// TwinCAT 3 PLC project PLC_Portale
// Title: TFPalletizer
// Author: Pugnaghi
// libraries:
//   Tc2_Math, * (Beckhoff Automation GmbH)
//   Tc2_MC2, * (Beckhoff Automation GmbH)
//   Tc2_MC2_Drive, * (Beckhoff Automation GmbH)
//   Tc2_Standard, * (Beckhoff Automation GmbH)
//   Tc2_SUPS, * (Beckhoff Automation GmbH)
//   Tc2_System, * (Beckhoff Automation GmbH)
//   Tc2_Utilities, * (Beckhoff Automation GmbH)
//   Tc3_Module, * (Beckhoff Automation GmbH)
//   Tc3_Standard, * (Beckhoff Automation GmbH)
//   TFDataLogger, * (Tecnoferrari)
//   TFInterpolazioneAssi, * (TecnoFerrari)
//   TFPLC, * (Tecnoferrari)
//   TF_CambioProduzioneLinea, * (Tecnoferrari)
//   TF_Ovem, * (Tecnoferrari)
// project tree:
//   Data types/AlbertoPruevas/BloqueFunciones/CalculoFormaciones/ Fb_CalculoCoordenadasFinalesFormacion.TcPOU, Fb_CalculoTodo180CoordenadasFinales.TcPOU, Fb_Fb_CalculoTodo0CoordenadasFinales.TcPOU
//   Data types/AlbertoPruevas/BloqueFunciones/ Fb_SensoresTasteggio.TcPOU
//   Data types/AlbertoPruevas/Enumeraciones/ E_Ul_RecogidaCaballete.TcDUT
//   Data types/AlbertoPruevas/Estructuras/Es_FormacionCaballete/EstructuraCaballetePiking/ ES_DatosPosCaballete.TcDUT, Es_PiezasCaballetePiking.TcDUT
//   Data types/AlbertoPruevas/Estructuras/Es_FormacionCaballete/ Es_CoordenadasCaballeteLadoA.TcDUT, Es_CoordenadasCaballeteLadoA_ladoB.TcDUT, Es_CoordenadasCaballeteLadoB.TcDUT, ES_dimensionPiezaLadoA_ladoB.TcDUT, Es_NumeroPiezasCaballete.TcDUT, ES_SpesoreLastra_A_B.TcDUT
//   Data types/AlbertoPruevas/Estructuras/ Es_Ingombro_PorPosicion.TcDUT (not stored), Es_LadosCaballete.TcDUT, Es_PiezasCaballete.TcDUT, ProgramaEjecucion.TcDUT
//   Data types/AlbertoPruevas/Funciones/FuncionesFormaciones/ Fun_CalculoCoordenadasFinalesFormacion.TcPOU
//   Data types/AlbertoPruevas/Funciones/ FunLadoTrabajoCaballete.TcPOU, Fun_NumeroPiezasLadoCaballete.TcPOU, Fun_PiezaLadoCaballete.TcPOU, Fun_SensoresTasteggio.TcPOU
//   Data types/DatiVari/EAP/ ST_EAPAxeState.TcDUT, ST_EAPCylinderState.TcDUT, ST_EAPMachineState.TcDUT, ST_EAPModuleState.TcDUT, ST_EAPOvemStatus.TcDUT, ST_EAPPinzaVenstoseStateComplete.TcDUT, ST_EAPPinzaVentoseDeviceState.TcDUT, ST_EAPStatoPortaleVisu.TcDUT
//   Data types/DatiVari/ e_StatoMacchinaWMS.TcDUT, e_SupportTypeAriostea.TcDUT, ST_HskFromSupervisor.TcDUT, ST_HskToSupervisor.TcDUT, ST_StatisticData.TcDUT, ST_SupervisorData.TcDUT
//   Data types/DatiVari/Workorder/ ST_DataWorkArea.TcDUT, ST_DimensionElement.TcDUT, ST_LayerData.TcDUT, ST_SlabData.TcDUT, ST_SupportData.TcDUT, ST_WorkOrder.TcDUT, ST_WorkOrder_Premium.TcDUT
//   Data types/Enum/ e_Disposizione_FTC_WA.TcTLEO, e_Disposizione_Postazioni.TcDUT, e_PosizionePinza.TcDUT, e_RiferimentoPostazione.TcTLEO, e_OrdinamentoPostazione.TcTLEO, e_StatoWorkOrder.TcDUT, e_Stato_Apprendimento.TcTLEO, e_Stato_ElementoLista.TcTLEO, e_Stato_Missione.TcTLEO, e_Stato_PickPoint.TcTLEO, e_Stato_Pareggiatura_Lastra.TcTLEO, e_Stato_LetturaBarCode.TcTLEO, e_Stato_Prodotto_Su_PickPoint.TcTLEO, e_Stato_Prelievo.TcTLEO, e_Stato_Ingombro_EE.TcTLEO, e_Stato_Layer.TcTLEO, e_Stato_Prodotto_Generico.TcTLEO, e_Stato_WAManager.TcTLEO, e_Priorita_PickPoint.TcTLEO, e_Stato_WorkArea.TcTLEO, e_Stato_ListaDiProduzione.TcTLEO, e_TipologiaAreaLaser.TcDUT, e_Tipologia_Rul_Prel.TcDUT, e_Tipo_Elemento_Da_Lavorare.TcDUT, e_Tipo_Magazzino_Falde.TcTLEO, e_Tipo_ChiusuraAsseK.TcTLEO, e_Tipo_Funzionamento.TcTLEO, e_Tipo_WorkArea.TcTLEO, e_Tipo_Ribaltino.TcTLEO, e_Tipo_PickPoint.TcTLEO, e_Tipo_Falda.TcTLEO, e_Tipo_Pallet.TcTLEO, e_Tipo_PresaEndEffector.TcTLEO, e_Tipo_Traiettoria.TcTLEO, e_Verso_Pallettizzatore.TcTLEO
//   Data types/Enum/Formatura/ e_TipologiaDeposito.TcDUT
//   Data types/Enum/Trasporti/ e_ElementZone.TcDUT, e_PosizioneRullieraMobile.TcDUT, e_StatoCentratura.TcDUT, e_TipoMacchinaTrasporti.TcDUT
//   Data types/LGV/ e_Tipo_Richiesta_LGV.TcTLEO, e_Stato_Richiesta_LGV_1.TcTLEO, LGV_Stato_Formatura.TcDUT, LGV_Stato_Pallettizzatore.TcDUT, LGV_Stato_Postazione.TcDUT, e_Stato_Operazione_LGV.TcTLEO
//   Data types/Nuove/ ST_OffsetAllDirection.TcDUT, TFMachinePalletizer_ListaProduzione_WAM_HMI.TcDUT, TFMachinePalletizer_WorkAreaTransport_State.TcDUT, TFMachinePalletizer_WorkPlacePointToPalletizer.TcDUT, TFMachinePalletizer_WorkPlacePointFromPalletizer.TcDUT, TFCodiciPerFormatura.TcDUT, TFError_WAM.TcDUT, TFMachinePalletizer_DataElementMP.TcDUT, TFMachinePalletizer_PinzaVentoseManCmd.TcDUT, TFMachinePalletizer_ApprendimentoQuota.TcDUT, TFMachinePalletizer_CoordinateApprendimento.TcDUT, TFMachinePalletizer_LatoApprendimento.TcDUT, TFMachinePalletizer_DataElement.TcDUT, TFMachinePalletizer_EndEffector.TcDUT, TFMachinePalletizer_BarCode.TcDUT, TFMachinePalletizer_ListaProduzione.TcDUT, TFMachinePalletizer_ListaProduzione_WAM.TcDUT, TFMachinePalletizer_OffsetElement.TcDUT, TFMachinePalletizer_PickPlaceParameters.TcDUT, TFMachinePalletizer_PinzaState.TcDUT, TFMAchinePalletizer_PinzaVentoseStatus.TcDUT, TFMachinePalletizer_PinzaVentose_OUT.TcDUT, TFMachinePalletizer_PlaceElement.TcDUT, TFMachinePalletizer_PlaceElementList.TcDUT, TFMachinePalletizer_WorkPickPointOffset.TcDUT, TFMachinePalletizer_WorkPickPoint_State.TcDUT, TFMachinePalletizer_WorkPickPointRoller_State_DaLinea.TcDUT, TFMachinePalletizer_WorkPickPointRoller_State_ALinea.TcDUT, TFMachinePalletizer_WorkPickPointStore_State.TcDUT, TFMachinePalletizer_WorkPickPointSlab.TcDUT, TF_CylinderState.TcDUT, TFMchinePalletizer_PinzaVentose_IN.TcDUT, TFPalletizerModules.TcDUT
//   Data types/Picking/ e_TypologySupDataPicking.TcDUT, ST_DataManualPicking.TcDUT, ST_WorkAreaDataPicking.TcDUT
//   Data types/Programmi Movimento/ TFModulePortaleStatus.TcDUT, AxHomingParameters.TcDUT, Ax_Palletizer_Basic_Parameters.TcDUT, Ax_Palletizer_Nominal_Parameters.TcDUT, GestioneEncoderEsterno.TcDUT, MissionStateCase.TcDUT, Module_Palletizer_Aspirazione_IN.TcDUT, Module_Palletizer_Aspirazione_ManCmd.TcDUT, Module_Palletizer_AX_OUT.TcDUT, Module_Palletizer_AX_IN.TcDUT, Ax_Program_Parameters.TcDUT, Descrittore_Programma.TcDUT, Ax_Palletizer_Parameters.TcDUT, Module_Palletizer_Aspirazione_OUT.TcDUT, OffsetSicurezzaIngombro.TcDUT, OffsetDistacco.TcDUT, Offset_Pass_Mode.TcDUT, Offset_Prelievi_Lenti.TcDUT, Offeset_Apprendimento.TcDUT, Offset_Sicurezza.TcDUT, Offset_Sicurezza_Anticipo_Movimenti.TcDUT, Overide_Dinamico.TcDUT, ProgrammaLog.TcDUT, Stato_Ciclo_Lavoro.TcDUT, StrutturaGenericaQuotaAssi.TcDUT, TFDimensioniPinza.TcDUT, TFMachinePalletizer_ModuleState.TcDUT, TFMachinePalletizer_MachineState.TcDUT, TFMachinePalletizer_VelocityOverride_TF.TcDUT, TFModulePalletizerRobot_Point_TF.TcDUT, TFModulePalletizerSTATUS_TF.TcDUT, TFTraiettoria.TcDUT, TFWorkAreaManager.TcDUT, Work_PickPoint_Dimension.TcDUT
//   Data types/ StatoPostazioneHMI.TcDUT, StatoLineaDepal.TcDUT, TFDatiDaLineaAPal.TcDUT, TFSlab.TcDUT
//   Data types/Programmi Movimento/Enum Programmi/ e_ProgrammiMovimentoX.TcTLEO, e_ProgrammiMovimentoJ.TcTLEO, e_ProgrammiMovimentoY.TcTLEO, e_ProgrammiMovimentoZ.TcTLEO
//   Data types/Scambio Dati Trasporti/ DUT_ArrayPacchi.TcDUT, DUT_Lista_Pacchi_In_Pila.TcDUT, DUT_Struttura_Dati_Pacco.TcDUT
//   Data types/Strutture Aggiornate/ TFMachinePalletizer_FormingForSlab.TcDUT, TFMachinePalletizer_Layer.TcDUT, TFMachinePalletizer_Mission.TcDUT, TFMachinePalletizer_Pallet.TcDUT, TFMachinePalletizer_PalletSlabOld.TcDUT, TFMachinePalletizer_WorkAreaState_VECCHIO.TcDUT, TFMachinePalletizer_WorkAreaState.TcDUT, TFMachinePalletizer_WorkArea.TcDUT, TFMachinePalletizer_WorkPickPoint.TcDUT, TFMachinePalletizer_WorkArea_VECCHIO.TcDUT, TFMachinePalletizer_FormingPack.TcDUT
//   Data types/TF/Aggiornate_20230504/ ST_BarcodeReaderReply.TcDUT, ST_BarcodeReaderRequest.TcDUT, ST_MachinePalletizerAxeManCmd.TcDUT, ST_MachinePalletizerAxeState.TcDUT, ST_MachinePalletizerMachineState.TcDUT, ST_MachinePalletizerModuleState.TcDUT, ST_MachinePalletizerPinzaDeviceState.TcDUT, ST_MachinePalletizerPinzaStateComplete.TcDUT, ST_MachinePalletizerPinzaVentoseManCmd.TcDUT, ST_StatoPostazioneHMI.TcDUT
//   Data types/TF/Barcode/ BarcodeStatus.TcDUT, InputDataLogic.TcDUT, InputKeyence.TcDUT, OutputDataLogic.TcDUT, OutputKeyence.TcDUT, StatusDataLogic.TcDUT, ST_ManCmdBarcode.TcDUT, TFDeviceBCStatus.TcDUT
//   Data types/TF/Handling/ TFHandlingPack.TcDUT
//   Data types/TF/Palletizer/ TFMachinePalletizer_AxeState_TF.TcDUT, TFMachinePalletizer_AxeState_weintek.TcDUT, TFMachinePalletizer_GatesAccess.TcDUT, TFMachinePalletizer_ManCmd.TcDUT, TFMachinePalletizer_ParametersFromHMI.TcDUT, TFMachinePalletizer_WorkAreaOffset.TcDUT, TFMachinePalletizer_WorkAreaSort.TcDUT, TFMachinePalletizer_WorkAreaZone.TcDUT, TFMachinePalletizer_WorkPickPointState_OLD.TcDUT, TFMachinePalletizer_WorkPPOffset.TcDUT, TFMachinePalletizer_Zone.TcDUT, TFModulePalletizerRobot_TCPPar.TcDUT, TFModulePalletizerRobot_Point.TcDUT, TFModulePalletizerRobot_ManCmd.TcDUT, TFMachinePalletizer_AxeParameters.TcDUT, TFMachinePalletizer_AxeManCmd.TcDUT, TFMachinePalletizer_AxeState.TcDUT, TFModulePalletizerRobot_AxisPar.TcDUT, TFMachinePalletizer_Forming_OLD.TcDUT, TFMachinePalletizer_FormingPack_OLD.TcDUT, TFMachinePalletizer_IN.TcDUT, TFMachinePalletizer_Layer_OLD.TcDUT, TFMachinePalletizer_OUT.TcDUT, TFMachinePalletizer_Pallet_OLD.TcDUT, TFMachinePalletizer_VelocityOverride.TcDUT, TFMachinePalletizer_WorkArea_OLD.TcDUT, TFMachinePalletizer_WorkFootprint.TcDUT, TFMachinePalletizer_WorkPickPoint_OLD.TcDUT, TFMachinePalletizer_WorkSpace.TcDUT, TFModulePalletizerRobot_Status.TcDUT, TFModulePalletizerRobot_IN.TcDUT, TFModulePalletizerRobot_OUT.TcDUT
//   Data types/TF/Rulliere/Macchina/ TFMachineTransportIN.TcDUT, TFMachineTransportManCmd.TcDUT, TFMachineTransportOUT.TcDUT
//   Data types/TF/Rulliere/Moduli/Cinghia/ TFCinghiaManCmd.TcDUT, TFCinghia_IN.TcDUT, TFBancoScelta_IN.TcDUT, TFCinghia_OUT.TcDUT, TFCinghiaParameters.TcDUT, TFBancoScelta_OUT.TcDUT, TFMoveParAXCinghia.TcDUT
//   Data types/TF/Rulliere/Moduli/RullieraPallet/ TFAxCentratoreManCmd.TcDUT, TFAxTraslazioneRulliera.TcDUT, TFCentratoreManCmd.TcDUT, TFCentratoreParameters.TcDUT, TFCentratoreStatus.TcDUT, TFCentratore_IN.TcDUT, TFCentratore_OUT.TcDUT, TFMoveParAXCentratore.TcDUT, TFMoveParAXRulliera.TcDUT, TFMoveParAXTraslazioneRulliera.TcDUT, TFRullieraManCmd.TcDUT, TFRullieraMobileManCmd.TcDUT, TFRullieraMobileStatus.TcDUT, TFRullieraParameters.TcDUT, TFRullieraStatus.TcDUT, TFRulliera_IN.TcDUT, TFRulliera_OUT.TcDUT, TFTraslazioneRullieraParameters.TcDUT, TFTraslazioneRulliera_IN.TcDUT
//   Data types/TF/Rulliere/Moduli/ TFAxManCmd.TcDUT, TFAxParameters.TcDUT, TFPortaStatus.TcDUT, TFPortaManCmd.TcDUT, TFGestioneFTC_Misura_OUT.TcDUT, TFBarcodeStatus.TcDUT, TFTransportModules.TcDUT, TFTransportModuleStatus.TcDUT
//   Data types/TF/Rulliere/ TFDimensionElement.TcDUT, TFMachinePalletizer_Pallet_Weintek.TcDUT, TFMachineTransportElement.TcDUT, TFMachineTransportElementWeintek.TcDUT, TFMachineTransport_GatesAccess.TcDUT
//   Global Variables/BarCode/ BarCODE.TcGVL
//   Global Variables/ Comandi_1.TcGVL, Safety.TcGVL, TFMachinesErrors.TcGVL, TFMachinePalletizerVariables.TcGVL, TFMachinePalletizerErrors.TcGVL, TFCmdStates.TcGVL, TFUpsVariables.TcGVL, TO_HMI.TcGVL
//   Global Variables/Configurazione Impianto/ Configurazione_Impianto.TcGVL
//   Global Variables/Errori/ Errori_BarCODE.TcGVL, Errori_CalcoloFormatura.TcGVL, Errori_WAManager.TcGVL
//   Global Variables/TFVariable/ DATA_LOGGER.TcGVL, Dati_Per_Linea.TcGVL, FROM_HMI_PAL.TcGVL, HMI_COMMAND_PAL.TcGVL, HMI_Formatura.TcGVL, IO_TRASPORTI.TcGVL, IO_Virtuali.TcGVL, LGV_Data.TcGVL, Picking.TcGVL, Pinza.TcGVL, QE_BORDO.TcGVL, QE_TERRA.TcGVL, Supervisor_Variable.TcGVL, TFGlobal.TcGVL, TFMotion_Program.TcGVL, TF_CambioProduzione.TcGVL
//   / GlobalTextList.TcGTLO, Plc_Portale.TcTTO, Visualization Manager.TcVMO (not stored)
//   POUs/Check/ CheckBounds.TcPOU, CheckDivDInt.TcPOU, CheckDivLInt.TcPOU, CheckDivLReal.TcPOU, CheckDivReal.TcPOU, CheckLRangeSigned.TcPOU, CheckLRangeUnsigned.TcPOU, CheckPointer.TcPOU, CheckRangeSigned.TcPOU, CheckRangeUnsigned.TcPOU
//   POUs/TFCicliDiLavoro/Lastre/Cicli Depallettizzatore/ TFCiclo_Deposito_Falda_Depal.TcPOU, TFCiclo_Deposito_Lastra_Depal.TcPOU, TFCiclo_Prelievo_Lastra_Depal.TcPOU
//   POUs/TFCicliDiLavoro/Lastre/Cicli di Deposito Lastre/ TFCiclo_Deposito_Falda.TcPOU, TFCiclo_Deposito_Lastra.TcPOU
//   POUs/TFCicliDiLavoro/Lastre/Cicli di Prelievo Lastre/ TFCiclo_Prelievo_Falda.TcPOU, TFCiclo_Prelievo_Lastra.TcPOU
//   POUs/TFCicliDiLavoro/Lastre/ TFCiclo_Di_Riposo_Lastre.TcPOU
//   POUs/TFCicliDiLavoro/ProgrammiMovimento/ TFProgramma_Ciclo_Falda_Lastre.TcPOU, TFProgramma_Ciclo_Lastra.TcPOU, TFProgramma_Ciclo_Riposo_Lastre.TcPOU
//   POUs/TFGateAccess/ TFGateAccess.TcPOU, TFGateAccessDoppiaMacchina.TcPOU, TFGateAccessNoStop.TcPOU
//   POUs/TFLGV/ GateAccessLGV.TcPOU, TFLGV.TcPOU, TFLGV_NEW.TcPOU
//   POUs/TFMachines/ TFMachinePalletizer_TF.TcPOU
//   POUs/TFMachines/Utility/ TFIsWorkflowError.TcPOU, TFIsWorkflowDisableOrEndedOrError.TcPOU, TFWorkflowsAllEnableOrDisable.TcPOU, TFWorkflowsCheckState.TcPOU
//   POUs/TFModules/DataBase/ Record_From_DB.TcDUT, StoredProcedureState.TcDUT, TFSPRicavaDatiDaBarcodeUDC.TcPOU, TFSPRichiestaIngressoMateriale.TcPOU, TFVerificaLetturaBarcodeConDatiDB.TcPOU
//   POUs/TFModules/Misurazione Ingresso/Keyence/ Keyence_LRTB2000C.TcPOU
//   POUs/TFModules/Misurazione Ingresso/ TFGestioneFTC_Misura.TcPOU, TFGestioneFTC_Misura_IN.TcDUT
//   POUs/TFModules/Moduli TF/ TFModulePalletizer_Aspirazione.TcPOU, TFModulePalletizer_AxJ_Lastre.TcPOU, TFModulePalletizer_Pinza.TcPOU, TFModulePalletizer_Pinza_mag.TcPOU, TFModulePalletizer_Pinza_2Ovem.TcPOU, TFModulePalletizer_Ax.TcPOU, TFModulePalletizer_Pinza_Semplice.TcPOU, TFProgramLogUpdate.TcPOU
//   POUs/TFModules/Utility/ TFClearAllCmdModulePinza.TcPOU, TFClearAllCmdModulePinzaCompleta.TcPOU, TFCylinder_ClearAllCommand.TcPOU, TFOVEMClearAllCommand.TcPOU, TFCylinder_HasCommand.TcPOU (excluded from build), TFPalletizerModulesCheckPowerActive.TcPOU, TFPalletizerModulesCommandSend.TcPOU, TFPalletizerModulesCheckState.TcPOU, TFPalletizerIsModuleError.TcPOU
//   POUs/TFPalletizerDataTF/FunzionePerNuovaGestioneTrasporti/ TFNumeroPacchiSuLinea.TcPOU, TFNumeroUltimi_N_TrasportiOccupati.TcPOU, TFPackCodePresenteInWAJolly.TcPOU (excluded from build), TFPackCodePresenteInZona.TcPOU (excluded from build), TFPackCodePresenteInZona_old.TcPOU (excluded from build)
//   POUs/TFPalletizerDataTF/NON_USATE/ TFCalcoliFuoriIngombriColonne.TcPOU (excluded from build), TFCalcoliFuoriIngombriColonne_old.TcPOU (excluded from build), TFCodicePaccoPresenteInFormatura.TcPOU (excluded from build), TFCodicePaccoPresenteInFormaturaAll.TcPOU (excluded from build), TFDepositoContinuoPalletConsentito.TcPOU (excluded from build), TFNumeroPacchiSuLinea_OLD.TcPOU (excluded from build), TFNumeroUltimi_N_TrasportiOccupati_OLD.TcPOU (excluded from build), TFPalletizerWorkAreaManagerTF.TcPOU (excluded from build), TFPalletizer_CalcolaCoordinataPrelievo_WorkArea.TcPOU (excluded from build), TFValutaFormatureMultipleAttivate.TcPOU (excluded from build), TFValutaSeFormaturaMista.TcPOU (excluded from build), TFWAconCodiceWPPPresente.TcPOU (excluded from build)
//   POUs/TFPalletizerDataTF/ TFCalcoliFuoriIngombri.TcPOU, TFCalcoliIngombroPinza_ConAsseK.TcPOU, TFCalcoloOverrideDinamico.TcPOU, TFCalcoloPuntiDiAnticipoDinamici.TcPOU, TFCalcoloVelocita.TcPOU, TFConsentiDepositoPaccoSuWA.TcPOU, TFCoppiaPinzaOk.TcPOU, TFControlloInterferenza.TcPOU, TFCalcoloTraiettoria_pacchi.TcPOU (excluded from build), TFFuoriIngombroVerticaleOK.TcPOU, TFPalletizerInPosizioneRiposo.TcPOU, TFPinzaInFuoriIngombroColonne_DirezioneX.TcPOU, TFValutaAssiInFinestraDiPassMode.TcPOU
//   POUs/TFPalletizerDataTF/Utility Varie/ TFAsseInFinestra.TcPOU, TFCalcolaFuoriIngombroY_oo.TcPOU, TFCalcolaNumeroPostazioneDXSX.TcPOU, TFCalcolaQuotaIngombroColonneLastre.TcPOU, TFCalcoliIngombroPinza.TcPOU, TFCalcoloIngombroOttimizzatoPinza.TcPOU, TFCalcoloTraiettoriaLastre.TcPOU, TFDirezioneAssePositiva.TcPOU, TFInverterV1000.TcPOU
//   POUs/TFPalletizerData/NON_USATE/ TFCheckPalletFull.TcPOU (excluded from build), TFClearWorkAreaStack.TcPOU (excluded from build), TFGetEnableCode.TcPOU (excluded from build), TFGetNearestWA.TcPOU, TFGripperNearTilter.TcPOU (excluded from build), TFLeastUsedCode.TcPOU (excluded from build), TFMostUsedCode.TcPOU (excluded from build), TFNextCommandToTilter.TcPOU (excluded from build), TFPackCodeOnWPP.TcPOU (excluded from build), TFPackCodePresentToJollyWorkArea.TcPOU (excluded from build), TFPackCodePresentToZone.TcPOU (excluded from build), TFPackOnPickPoint.TcPOU (excluded from build), TFPalletizerCheckPalletLayerCode.TcPOU (excluded from build), TFPalletizerGetFormingFromCode.TcPOU (excluded from build), TFPalletizerGetUnassignedCode.TcPOU (excluded from build), TFPalletizerGetWAFromTypeCode.TcPOU (excluded from build), TFPalletizerGetWPPFromPackCode.TcPOU (excluded from build), TFPalletizerIsCodeAssigned.TcPOU (excluded from build), TFPalletizerIsFormingAssigned.TcPOU (excluded from build), TFPalletizerIsStackAvailable.TcPOU (excluded from build), TFPalletizerPackValidation.TcPOU (excluded from build), TFRefreshUsedCode.TcPOU (excluded from build), TFWorkareaConPacchiComplete.TcPOU (excluded from build)
//   POUs/TFPalletizerData/ TFCheckPalletPresence.TcPOU, RestoringCWA.TcPOU, TFCheckLayerPresence.TcPOU, TFClearWorkArea.TcPOU, TFClearWorkAreaArray.TcPOU, TFClearWorkAreaStateSlab.TcPOU, TFPalletizerIsWorkAreaIntoZone.TcPOU (excluded from build)
//   POUs/TFPalletizerData_Lastre/Formatura/ Calcolo_Formatura_Completa.TcPOU, Calcolo_Formatura_Completa_24_10_2025.TcPOU
//   POUs/TFPalletizerData_Lastre/Formatura/FuncionesFormacionParaquitar/ Calcolo_Formatura_CompletaNew.TcPOU (not stored), Calcolo_Formatura_Completa_Back.TcPOU, Calcolo_Formatura_Completa_Backup16_10_25.TcPOU (not stored)
//   POUs/TFPalletizerData_Lastre/Formatura/Utility/CSV read_write in text mode/ P_TextModeRead.TcPOU, P_TextModeWrite.TcPOU
//   POUs/TFPalletizerData_Lastre/ TFAggiuntaSupportoManuale.TcPOU, TFClearWorkAreaBCRead.TcPOU, TFClearApprendimento.TcPOU, TFGetEnableCode_Lastre.TcPOU, TFPalletizerGestione_PickPoint_Rulliere.TcPOU, TFPalletizerGetFormingFromCodeSlab.TcPOU, TFPalletizerPackValidationSlab.TcPOU, TFPalletizerPickRollerPriority.TcPOU, TFPalletizer_CalcolaCoordinataPrelievo_PickPoint.TcPOU, TFPalletizerGetNumPickPointForLayerCode.TcPOU, TFPalletizerGetWPPFromLastraCode.TcPOU, TFPalletizerWorkAreaManagerTF_Lastre.TcPOU, TFWAM_CreaMissione_DepPrelElemento.TcPOU, TFWAM_RicavaListaInLavoro.TcPOU
//   POUs/TFVisuText/ HandlingModulesCmd.TcTLO, HandlingModulesState.TcTLO, KPickMode.TcTLO, KUnLoadMode.TcTLO, KPickType.TcTLO, KLoadMode.TcTLO, KProduct.TcTLO, KPlaceMode.TcTLO, MissionText.TcTLO, PXExitYesNo.TcTLO, WorkAreaLearn.TcTLO, WorkAreaLGVLetIn.TcTLO, WorkAreaLGVReq.TcTLO, WorkAreaStatePN.TcTLO, WorkAreaTypology.TcTLO, WorkAreaYesNo.TcTLO, WorkAreaState.TcTLO
//   POUs/TFPrograms/ TFMachinePalletizerMain.TcPOU, TFUps.TcPOU (excluded from build)
//   Visualizations/ Pallettizzatore.TcVIS, Stato_Missione.TcTLO, Stato_WAM.TcTLO
// real-time tasks:
//   TASK PlcTask_Portale: cycle T#1ms, priority 6, ADS port 351
// motion (NC):
//   TASK NC-Task 1 SAF: cycle T#4ms, priority 8, ADS port 501
//   TASK NC-Task 1 SVB: cycle T#4ms, priority 10, ADS port 511
//   AXIS X (id 1)
//     Dynamic: AccelerationMaximum=5000, DecelerationMaximum=5000, Acceleration=5000, Deceleration=5000, Jerk=5000
//     Velo: RefSearch=100, RefSync=10, FastManual=200, Fast=3005.36226499422, Maximum=2500
//     OtherSettings: AllowMotionCmdToSlave=true, PulseDistanceNeg=0.1
//     encoder EncType=19
//       EncPara: ScaleFactorNumerator=37.369, ScaleFactorDenominator=65536, Offset=-1080.65753173828, EncMode=3, MaxCount=#xffffffff
//         FilterTime: TVelo=0, TAcc=0
//         SoftEndMinControl: Enable=true, Range=0.5
//         SoftEndMaxControl: Enable=true, Range=33345
//         Inc: RefSearchInverse=true, RefSyncInverse=false
//     drive DrvType=16
//       DrvPara: MaxCount=#xffffffff
//         Analog: VeloReferenz=2500, TorqueSetpointScale=10, ScaleFactorActTorque=1
//         TimeComp: TaskDelayCycles=1
//     controller CtrType=1
//       CtrPara: PriorControlFactor=1
//         PosDiffControl: Range=500, Time=0.05
//         Observer: BandWidth=20
//   AXIS Y (id 2)
//     Dynamic: AccelerationMaximum=2924.81, DecelerationMaximum=2924.81, Acceleration=1882.24, Deceleration=1882.24, Jerk=5046.78
//     Velo: RefSearch=100, RefSync=2, SlowManual=20, FastManual=100, Fast=1949.87615168843, Maximum=2600
//     OtherSettings: AllowMotionCmdToSlave=true, PulseDistancePos=50
//     encoder EncType=19
//       EncPara: ScaleFactorNumerator=27.7398016228, ScaleFactorDenominator=65536, Offset=38938.6948199463, Inverse=true, MaxCount=#xffffffff
//         FilterTime: TVelo=0, TAcc=0
//         SoftEndMinControl: Enable=true, Range=445
//         SoftEndMaxControl: Enable=true, Range=3300
//         Inc: RefSearchInverse=true, RefSyncInverse=false
//     drive DrvType=16
//       DrvPara: Inverse=true, MaxCount=#xffffffff
//         Analog: VeloReferenz=2600, TorqueSetpointScale=10, ScaleFactorActTorque=1
//         TimeComp: TaskDelayCycles=1
//     controller CtrType=1
//       CtrPara: PriorControlFactor=1
//         PosDiffControl: Range=50
//         Observer: BandWidth=20
//   AXIS Z (id 3)
//     Dynamic: AccelerationMaximum=4000, DecelerationMaximum=4000, Acceleration=6000, Deceleration=6000, Jerk=10000
//     Velo: RefSearch=24.9356063175, RefSync=24.9356063175, FastManual=748.068189525, Fast=2493.56063175, Maximum=520
//     OtherSettings: AllowMotionCmdToSlave=true
//     encoder EncType=19
//       EncPara: ScaleFactorNumerator=6.908, ScaleFactorDenominator=65536, Offset=-5733.66098022461, EncMode=3, MaxCount=#xffffffff
//         FilterTime: TVelo=0, TAcc=0
//         SoftEndMinControl: Enable=true, Range=20
//         SoftEndMaxControl: Enable=true, Range=1926
//     drive DrvType=16
//       DrvPara: MaxCount=#xffffffff
//         Analog: VeloReferenz=520, TorqueSetpointScale=10, ScaleFactorActTorque=1
//         TimeComp: TaskDelayCycles=1
//     controller CtrType=1
//       CtrPara: PriorControlFactor=1
//         PosDiffControl: Range=100
//         Observer: BandWidth=20
//   AXIS J (id 22)
//     General: UnitName=°
//     Dynamic: AccelerationMaximum=3000, DecelerationMaximum=3000, Acceleration=346, Deceleration=346, Jerk=819.973
//     Velo: RefSearch=5, RefSync=1, SlowManual=5, FastManual=10, Fast=200.249663085938, Maximum=200
//     OtherSettings: AllowMotionCmdToSlave=true, PulseDistanceNeg=1
//     encoder EncType=19
//       EncPara: ScaleFactorNumerator=1.44, ScaleFactorDenominator=65536, Offset=-917.549625244141, Inverse=true, MaxCount=#xffffffff
//         SoftEndMinControl: Enable=true, Range=-1
//         SoftEndMaxControl: Enable=true, Range=181.600006103516
//         Inc: RefSearchInverse=true, RefSyncInverse=false
//     drive DrvType=16
//       DrvPara: Inverse=true, MaxCount=#xffffffff
//         Analog: VeloReferenz=220, TorqueSetpointScale=10, ScaleFactorActTorque=1
//         TimeComp: TaskDelayCycles=1
//     controller CtrType=1
//       CtrPara: PriorControlFactor=1
//         PosDiffControl: Range=20
//         Observer: BandWidth=20
// I/O:
//   DEVICE Dispositivo 3 (EtherCAT), AmsNetId 0.0.0.0.4.1
//     AP200_1 (EK1100) [EK1100 EtherCAT Coupler (2A E-Bus)]
//       AP200 2 (EL1809) [EL1809 16Ch. Dig. Input 24V, 3ms]
//       AP200_3 (EL1904) [EL1904, 4 Ch. Safety Input 24V, TwinSAFE]
//         modules: Module 1 (FSOES)
//       AP200_4 (EL1904) [EL1904, 4 Ch. Safety Input 24V, TwinSAFE]
//         modules: Module 1 (FSOES)
//       AP200_5 (EL1809) [EL1809 16Ch. Dig. Input 24V, 3ms]
//       AP200_6 (EL1904) [EL1904, 4 Ch. Safety Input 24V, TwinSAFE]
//         modules: Module 1 (FSOES)
//       AP200_7 (EL1904) [EL1904, 4 Ch. Safety Input 24V, TwinSAFE]
//         modules: Module 1 (FSOES)
//       AP200_8 (EL1809) [EL1809 16Ch. Dig. Input 24V, 3ms]
//       AP200_9 (EL1904) [EL1904, 4 Ch. Safety Input 24V, TwinSAFE]
//         modules: Module 1 (FSOES)
//       AP200_10 (EL1904) [EL1904, 4 Ch. Safety Input 24V, TwinSAFE]
//         modules: Module 1 (FSOES)
//       AP201_1 (EL9410) [EL9410 E-Bus Power Supplier  (Diagnostics)]
//       AP201_2 (EL1904) [EL1904, 4 Ch. Safety Input 24V, TwinSAFE]
//         modules: Module 1 (FSOES)
//       AP201_3 (EL1809) [EL1809 16Ch. Dig. Input 24V, 3ms]
//       AP202_4 (EL6910) [EL6910, TwinSAFE PLC]
//       AP201_4 (EL2809) [EL2809 16Ch. Dig. Output 24V, 0.5A]
//       AP201_5 (EL2904) [EL2904, 4 Ch. Safety Output 24V, 0.5A, TwinSAFE]
//         modules: Module 1 (FSOES), Module 2 (DO)
//       AP201_6 (EL2809) [EL2809 16Ch. Dig. Output 24V, 0.5A]
//       AP202_2 (EL1904) [EL1904, 4 Ch. Safety Input 24V, TwinSAFE]
//         modules: Module 1 (FSOES)
//       AP202_1 (EL9410) [EL9410 E-Bus Power Supplier  (Diagnostics)]
//       AP202_3 (EL1904) [EL1904, 4 Ch. Safety Input 24V, TwinSAFE]
//         modules: Module 1 (FSOES)
//       AP202_5 (EL1904) [EL1904, 4 Ch. Safety Input 24V, TwinSAFE]
//         modules: Module 1 (FSOES)
//       AP202_6 (EL1904) [EL1904, 4 Ch. Safety Input 24V, TwinSAFE]
//         modules: Module 1 (FSOES)
//       AP202_7 (EL9011) [EL9011 End Terminal]
//     AsseX (MOVI-C MOVIDRIVE CiA402) [MOVI-C MOVIDRIVE CiA402]
//       modules: Module 1 (Switching modes of operation), Module 2 (FSoE Safety IO 48 bit), Module 4 (FSoE empty)
//     AsseY (MOVI-C MOVIDRIVE CiA402) [MOVI-C MOVIDRIVE CiA402]
//       modules: Module 1 (Switching modes of operation), Module 2 (FSoE Safety IO 48 bit)
//     AsseZ (MOVI-C MOVIDRIVE CiA402) [MOVI-C MOVIDRIVE CiA402]
//       modules: Module 1 (Switching modes of operation), Module 2 (FSoE Safety IO 48 bit)
//     AsseJ (MOVI-C MOVIDRIVE CiA402) [MOVI-C MOVIDRIVE CiA402]
//       modules: Module 1 (Switching modes of operation), Module 2 (FSoE Safety IO 48 bit)
//     Ciabatta IFM Pinza K515 (ifm IO-Link Master AL1332)_1
//     Ciabatta IFM Pinza K516 (ifm IO-Link Master AL1332)_2
// variable links:
//   Device 3 (EtherCAT) <-> Device 3 (EtherCAT)/AP200_1 (EK1100)/AP200_10 (EL1904)
//     AP200_1 (EK1100)/AP202_4 (EL6910)/ConnectionInputs/IO.AP200_10 (EL1904) - Module 1 (FSOES)_284 TxPDO <-> Module 1 (FSOES)/RxPDO/FSOE
//     AP200_1 (EK1100)/AP202_4 (EL6910)/ConnectionOutputs/IO.AP200_10 (EL1904) - Module 1 (FSOES)_284 RxPDO <-> Module 1 (FSOES)/TxPDO/FSOE
//   Device 3 (EtherCAT) <-> Device 3 (EtherCAT)/AP200_1 (EK1100)/AP200_3 (EL1904)
//     AP200_1 (EK1100)/AP202_4 (EL6910)/ConnectionInputs/IO.AP200_3 (EL1904) - Module 1 (FSOES)_279 TxPDO <-> Module 1 (FSOES)/RxPDO/FSOE
//     AP200_1 (EK1100)/AP202_4 (EL6910)/ConnectionOutputs/IO.AP200_3 (EL1904) - Module 1 (FSOES)_279 RxPDO <-> Module 1 (FSOES)/TxPDO/FSOE
//   Device 3 (EtherCAT) <-> Device 3 (EtherCAT)/AP200_1 (EK1100)/AP200_4 (EL1904)
//     AP200_1 (EK1100)/AP202_4 (EL6910)/ConnectionInputs/IO.AP200_4 (EL1904) - Module 1 (FSOES)_280 TxPDO <-> Module 1 (FSOES)/RxPDO/FSOE
//   Device 3 (EtherCAT) <-> Device 3 (EtherCAT)/AP200_1 (EK1100)/AP200_6 (EL1904)
//     AP200_1 (EK1100)/AP202_4 (EL6910)/ConnectionInputs/IO.AP200_6 (EL1904) - Module 1 (FSOES)_281 TxPDO <-> Module 1 (FSOES)/RxPDO/FSOE
//   Device 3 (EtherCAT) <-> Device 3 (EtherCAT)/AP200_1 (EK1100)/AP200_9 (EL1904)
//     AP200_1 (EK1100)/AP202_4 (EL6910)/ConnectionOutputs/IO.AP200_9 (EL1904) - Module 1 (FSOES)_283 RxPDO <-> Module 1 (FSOES)/TxPDO/FSOE
//   Device 3 (EtherCAT) <-> Device 3 (EtherCAT)/AP200_1 (EK1100)/AP201_2 (EL1904)
//     AP200_1 (EK1100)/AP202_4 (EL6910)/ConnectionInputs/IO.AP201_2 (EL1904) - Module 1 (FSOES)_285 TxPDO <-> Module 1 (FSOES)/RxPDO/FSOE
//   Device 3 (EtherCAT) <-> Device 3 (EtherCAT)/AP200_1 (EK1100)/AP202_2 (EL1904)
//     AP200_1 (EK1100)/AP202_4 (EL6910)/ConnectionOutputs/IO.AP202_2 (EL1904) - Module 1 (FSOES)_287 RxPDO <-> Module 1 (FSOES)/TxPDO/FSOE
//   Device 3 (EtherCAT) <-> Device 3 (EtherCAT)/AP200_1 (EK1100)/AP202_4 (EL6910)
//     AP200_1 (EK1100)/AP200_4 (EL1904)/Module 1 (FSOES)/TxPDO/FSOE <-> ConnectionOutputs/IO.AP200_4 (EL1904) - Module 1 (FSOES)_280 RxPDO
//     AP200_1 (EK1100)/AP200_6 (EL1904)/Module 1 (FSOES)/TxPDO/FSOE <-> ConnectionOutputs/IO.AP200_6 (EL1904) - Module 1 (FSOES)_281 RxPDO
//     AP200_1 (EK1100)/AP200_7 (EL1904)/Module 1 (FSOES)/TxPDO/FSOE <-> ConnectionOutputs/IO.AP200_7 (EL1904) - Module 1 (FSOES)_282 RxPDO
//     AP200_1 (EK1100)/AP201_2 (EL1904)/Module 1 (FSOES)/TxPDO/FSOE <-> ConnectionOutputs/IO.AP201_2 (EL1904) - Module 1 (FSOES)_285 RxPDO
//     AP200_1 (EK1100)/AP201_5 (EL2904)/Module 1 (FSOES)/TxPDO/FSOE <-> ConnectionOutputs/IO.AP201_5 (EL2904) - Module 1 (FSOES)_286 RxPDO
//     AP200_1 (EK1100)/AP202_3 (EL1904)/Module 1 (FSOES)/TxPDO/FSOE <-> ConnectionOutputs/IO.AP202_3 (EL1904) - Module 1 (FSOES)_288 RxPDO
//     AP200_1 (EK1100)/AP202_6 (EL1904)/Module 1 (FSOES)/TxPDO/FSOE <-> ConnectionOutputs/IO.AP202_6 (EL1904) - Module 1 (FSOES)_290 RxPDO
//     AP200_1 (EK1100)/AP200_7 (EL1904)/Module 1 (FSOES)/RxPDO/FSOE <-> ConnectionInputs/IO.AP200_7 (EL1904) - Module 1 (FSOES)_282 TxPDO
//     AP200_1 (EK1100)/AP200_9 (EL1904)/Module 1 (FSOES)/RxPDO/FSOE <-> ConnectionInputs/IO.AP200_9 (EL1904) - Module 1 (FSOES)_283 TxPDO
//     AP200_1 (EK1100)/AP201_5 (EL2904)/Module 1 (FSOES)/RxPDO/FSOE <-> ConnectionInputs/IO.AP201_5 (EL2904) - Module 1 (FSOES)_286 TxPDO
//     AP200_1 (EK1100)/AP202_2 (EL1904)/Module 1 (FSOES)/RxPDO/FSOE <-> ConnectionInputs/IO.AP202_2 (EL1904) - Module 1 (FSOES)_287 TxPDO
//     AP200_1 (EK1100)/AP202_3 (EL1904)/Module 1 (FSOES)/RxPDO/FSOE <-> ConnectionInputs/IO.AP202_3 (EL1904) - Module 1 (FSOES)_288 TxPDO
//     AP200_1 (EK1100)/AP202_6 (EL1904)/Module 1 (FSOES)/RxPDO/FSOE <-> ConnectionInputs/IO.AP202_6 (EL1904) - Module 1 (FSOES)_290 TxPDO
//     AsseJ (MOVI-C MOVIDRIVE CiA402)/Module 2 (FSoE Safety IO 48 bit)/FSoE Safety Inputs 48 bit/FSOE <-> ConnectionOutputs/ZonaPallet.AsseJ (MOVI-C MOVIDRIVE CiA402) - Module 2 (FSoE Safety IO 48 bit)_278 RxPDO
//     AsseX (MOVI-C MOVIDRIVE CiA402)/Module 2 (FSoE Safety IO 48 bit)/FSoE Safety Inputs 48 bit/FSOE <-> ConnectionOutputs/ZonaPallet.AsseX (MOVI-C MOVIDRIVE CiA402) - Module 2 (FSoE Safety IO 48 bit)_275 RxPDO
//     AsseX (MOVI-C MOVIDRIVE CiA402)/Module 2 (FSoE Safety IO 48 bit)/FSoE Safety Outputs 48 bit/FSOE <-> ConnectionInputs/ZonaPallet.AsseX (MOVI-C MOVIDRIVE CiA402) - Module 2 (FSoE Safety IO 48 bit)_275 TxPDO
//     AsseZ (MOVI-C MOVIDRIVE CiA402)/Module 2 (FSoE Safety IO 48 bit)/FSoE Safety Outputs 48 bit/FSOE <-> ConnectionInputs/ZonaPallet.AsseZ (MOVI-C MOVIDRIVE CiA402) - Module 2 (FSoE Safety IO 48 bit)_277 TxPDO
//   Device 3 (EtherCAT) <-> Device 3 (EtherCAT)/AP200_1 (EK1100)/AP202_5 (EL1904)
//     AP200_1 (EK1100)/AP202_4 (EL6910)/ConnectionInputs/IO.AP202_5 (EL1904) - Module 1 (FSOES)_289 TxPDO <-> Module 1 (FSOES)/RxPDO/FSOE
//     AP200_1 (EK1100)/AP202_4 (EL6910)/ConnectionOutputs/IO.AP202_5 (EL1904) - Module 1 (FSOES)_289 RxPDO <-> Module 1 (FSOES)/TxPDO/FSOE
//   Device 3 (EtherCAT) <-> Device 3 (EtherCAT)/AsseJ (MOVI-C MOVIDRIVE CiA402)
//     AP200_1 (EK1100)/AP202_4 (EL6910)/ConnectionInputs/ZonaPallet.AsseJ (MOVI-C MOVIDRIVE CiA402) - Module 2 (FSoE Safety IO 48 bit)_278 TxPDO <-> Module 2 (FSoE Safety IO 48 bit)/FSoE Safety Outputs 48 bit/FSOE
//   Device 3 (EtherCAT) <-> Device 3 (EtherCAT)/AsseY (MOVI-C MOVIDRIVE CiA402)
//     AP200_1 (EK1100)/AP202_4 (EL6910)/ConnectionInputs/ZonaPallet.AsseY (MOVI-C MOVIDRIVE CiA402) - Module 2 (FSoE Safety IO 48 bit)_276 TxPDO <-> Module 2 (FSoE Safety IO 48 bit)/FSoE Safety Outputs 48 bit/FSOE
//     AP200_1 (EK1100)/AP202_4 (EL6910)/ConnectionOutputs/ZonaPallet.AsseY (MOVI-C MOVIDRIVE CiA402) - Module 2 (FSoE Safety IO 48 bit)_276 RxPDO <-> Module 2 (FSoE Safety IO 48 bit)/FSoE Safety Inputs 48 bit/FSOE
//   Device 3 (EtherCAT) <-> Device 3 (EtherCAT)/AsseZ (MOVI-C MOVIDRIVE CiA402)
//     AP200_1 (EK1100)/AP202_4 (EL6910)/ConnectionOutputs/ZonaPallet.AsseZ (MOVI-C MOVIDRIVE CiA402) - Module 2 (FSoE Safety IO 48 bit)_277 RxPDO <-> Module 2 (FSoE Safety IO 48 bit)/FSoE Safety Inputs 48 bit/FSOE
//   PLC_Portale/PLC_Portale Instance <-> Device 3 (EtherCAT)/AP200_1 (EK1100)/AP200 2 (EL1809)
//     Plc_Portale Inputs/.I_AP200_2[{1..16}] <-> Channel {1..16}/Input  (16 links)
//   PLC_Portale/PLC_Portale Instance <-> Device 3 (EtherCAT)/AP200_1 (EK1100)/AP200_10 (EL1904)
//     Plc_Portale Inputs/.I_AP200_10[{1..4}] <-> Module 1 (FSOES)/TxPDO/FSOE/InputChannel{1..4}  (4 links)
//   PLC_Portale/PLC_Portale Instance <-> Device 3 (EtherCAT)/AP200_1 (EK1100)/AP200_3 (EL1904)
//     Plc_Portale Inputs/.I_AP200_3[{1..4}] <-> Module 1 (FSOES)/TxPDO/FSOE/InputChannel{1..4}  (4 links)
//   PLC_Portale/PLC_Portale Instance <-> Device 3 (EtherCAT)/AP200_1 (EK1100)/AP200_4 (EL1904)
//     Plc_Portale Inputs/.I_AP200_4[{1..4}] <-> Module 1 (FSOES)/TxPDO/FSOE/InputChannel{1..4}  (4 links)
//   PLC_Portale/PLC_Portale Instance <-> Device 3 (EtherCAT)/AP200_1 (EK1100)/AP200_5 (EL1809)
//     Plc_Portale Inputs/.I_AP200_5[{1..16}] <-> Channel {1..16}/Input  (16 links)
//   PLC_Portale/PLC_Portale Instance <-> Device 3 (EtherCAT)/AP200_1 (EK1100)/AP200_6 (EL1904)
//     Plc_Portale Inputs/.I_AP200_6[{1..4}] <-> Module 1 (FSOES)/TxPDO/FSOE/InputChannel{1..4}  (4 links)
//   PLC_Portale/PLC_Portale Instance <-> Device 3 (EtherCAT)/AP200_1 (EK1100)/AP200_7 (EL1904)
//     Plc_Portale Inputs/.I_AP200_7[{1..4}] <-> Module 1 (FSOES)/TxPDO/FSOE/InputChannel{1..4}  (4 links)
//   PLC_Portale/PLC_Portale Instance <-> Device 3 (EtherCAT)/AP200_1 (EK1100)/AP200_8 (EL1809)
//     Plc_Portale Inputs/.I_AP200_8[{1..16}] <-> Channel {1..16}/Input  (16 links)
//   PLC_Portale/PLC_Portale Instance <-> Device 3 (EtherCAT)/AP200_1 (EK1100)/AP200_9 (EL1904)
//     Plc_Portale Inputs/.I_AP200_9[{1..4}] <-> Module 1 (FSOES)/TxPDO/FSOE/InputChannel{1..4}  (4 links)
//   PLC_Portale/PLC_Portale Instance <-> Device 3 (EtherCAT)/AP200_1 (EK1100)/AP201_2 (EL1904)
//     Plc_Portale Inputs/.I_AP201_2[{1..4}] <-> Module 1 (FSOES)/TxPDO/FSOE/InputChannel{1..4}  (4 links)
//   PLC_Portale/PLC_Portale Instance <-> Device 3 (EtherCAT)/AP200_1 (EK1100)/AP201_3 (EL1809)
//     Plc_Portale Inputs/.I_AP201_3[{1..16}] <-> Channel {1..16}/Input  (16 links)
//   PLC_Portale/PLC_Portale Instance <-> Device 3 (EtherCAT)/AP200_1 (EK1100)/AP201_4 (EL2809)
//     Plc_Portale Outputs/.O_AP201_4[{1..16}] <-> Channel {1..16}/Output  (16 links)
//   PLC_Portale/PLC_Portale Instance <-> Device 3 (EtherCAT)/AP200_1 (EK1100)/AP201_6 (EL2809)
//     Plc_Portale Outputs/.O_AP201_6[{1..16}] <-> Channel {1..16}/Output  (16 links)
//   PLC_Portale/PLC_Portale Instance <-> Device 3 (EtherCAT)/AP200_1 (EK1100)/AP202_2 (EL1904)
//     Plc_Portale Inputs/.I_AP202_2[{1..4}] <-> Module 1 (FSOES)/TxPDO/FSOE/InputChannel{1..4}  (4 links)
//   PLC_Portale/PLC_Portale Instance <-> Device 3 (EtherCAT)/AP200_1 (EK1100)/AP202_3 (EL1904)
//     Plc_Portale Inputs/.I_AP202_3[{1..4}] <-> Module 1 (FSOES)/TxPDO/FSOE/InputChannel{1..4}  (4 links)
//   PLC_Portale/PLC_Portale Instance <-> Device 3 (EtherCAT)/AP200_1 (EK1100)/AP202_4 (EL6910)
//     Plc_Portale Inputs/.I_MarciaOK <-> StandardInputs/IO.O_MarciaOkPortale_240
//     Plc_Portale Inputs/.I_RicevitoreConsensoVeicolo[1] <-> StandardInputs/IO.O_RicevitoreConsVeicolo1_158
//     Plc_Portale Inputs/.I_RicevitoreConsensoVeicolo[2] <-> StandardInputs/IO.O_RicevitoreConsVeicolo2_157
//     Plc_Portale Inputs/.I_RicevitoreConsensoVeicolo[3] <-> StandardInputs/IO.O_RicevitoreConsVeicolo3_156
//     Plc_Portale Inputs/.I_RicevitoreConsensoVeicolo[4] <-> StandardInputs/IO.O_RicevitoreConsVeicolo4_155
//     Plc_Portale Inputs/.I_RicevitoreConsensoVeicolo[5] <-> StandardInputs/IO.O_RicevitoreConsVeicolo5_154
//     Plc_Portale Inputs/.I_RicevitoreConsensoVeicolo[6] <-> StandardInputs/IO.O_RicevitoreConsVeicolo6_153
//     Plc_Portale Inputs/.I_RicevitoreConsensoVeicolo[7] <-> StandardInputs/IO.O_RicevitoreConsVeicolo7_291
//     Plc_Portale Inputs/.I_RicevitoreConsensoVeicolo[8] <-> StandardInputs/IO.O_RicevitoreConsVeicolo8_292
//     Plc_Portale Inputs/.I_SafetyCOMERR <-> StandardInputs/IO.O_SafetyCOMERR_54
//     Plc_Portale Inputs/.I_SafetyFBERR <-> StandardInputs/IO.O_SafetyFBERR_55
//     Plc_Portale Inputs/.I_SafetyOUTERR <-> StandardInputs/IO.O_SafetyOUTERR_57
//     Plc_Portale Inputs/.I_SafetyStateBarrierCentroDXPal <-> Function Block Info Data/ZonaPallet.BarrieraDX.BarrieraDXCentro Info Data/State
//     Plc_Portale Inputs/.I_SafetyStateBarrierCentroSXPal <-> Function Block Info Data/ZonaPallet.BarrieraSX.BarrieraSXCentro Info Data/State
//     Plc_Portale Inputs/.I_SafetyStateBarrierDXPal <-> Function Block Info Data/ZonaPallet.BarrieraDX.BarrieraDX Info Data/State
//     Plc_Portale Inputs/.I_SafetyStateBarrierKarv <-> Function Block Info Data/ZonaPallet.Karv.BarrieraKarv Info Data/State
//     Plc_Portale Inputs/.I_SafetyStateBarrierSXPal <-> Function Block Info Data/ZonaPallet.BarrieraSX.BarrieraSX Info Data/State
//     Plc_Portale Inputs/.I_SafetyStateEmergenza_PS306_307 <-> Function Block Info Data/ZonaPallet.Funghi.FunghiEmergenza306_307 Info Data/State
//     Plc_Portale Inputs/.I_SafetyStateEmergenza_PS308_309 <-> Function Block Info Data/ZonaPallet.Funghi.FunghiEmergenza308_309 Info Data/State
//     Plc_Portale Inputs/.I_SafetyStateEmergenze_Generali <-> Function Block Info Data/Globali.FunghiGlobali.GeneraleFunghi Info Data/State
//     Plc_Portale Outputs/.EnableGroupPortSafety <-> StandardOutputs/Globali.GroupPort_RunStop_303
//     Plc_Portale Outputs/.EnableGroupPortSafety <-> StandardOutputs/IO.GroupPort_RunStop_304
//     Plc_Portale Outputs/.EnableGroupPortSafety <-> StandardOutputs/ZonaPallet.GroupPort_RunStop_305
//     Plc_Portale Outputs/.O_AbilitazioneMarcia <-> StandardOutputs/IO.I_EnableMarciaPalettizzatore_26
//     Plc_Portale Outputs/.O_OverrideSoftwareBarriere_Pal <-> StandardOutputs/IO.I_OverrideBarrierePalett_41
//     Plc_Portale Outputs/.O_ResetACKAzionamenti <-> StandardOutputs/ZonaPallet.I_ErrorAcknowledgementAzionamenti_34
//     Plc_Portale Outputs/.O_Reset_Plc_Sicurezza <-> StandardOutputs/Globali.ErrorAcknowledgement_32
//     Plc_Portale Outputs/.O_Reset_Plc_Sicurezza <-> StandardOutputs/IO.ErrorAcknowledgement_1
//     Plc_Portale Outputs/.O_Reset_Plc_Sicurezza <-> StandardOutputs/ZonaPallet.ErrorAcknowledgement_25
//   PLC_Portale/PLC_Portale Instance <-> Device 3 (EtherCAT)/AP200_1 (EK1100)/AP202_5 (EL1904)
//     Plc_Portale Inputs/.I_AP202_5[{1..4}] <-> Module 1 (FSOES)/TxPDO/FSOE/InputChannel{1..4}  (4 links)
//   PLC_Portale/PLC_Portale Instance <-> Device 3 (EtherCAT)/AP200_1 (EK1100)/AP202_6 (EL1904)
//     Plc_Portale Inputs/.I_AP202_6[{1..4}] <-> Module 1 (FSOES)/TxPDO/FSOE/InputChannel{1..4}  (4 links)
//   PLC_Portale/PLC_Portale Instance <-> Device 3 (EtherCAT)/AsseJ (MOVI-C MOVIDRIVE CiA402)
//     Plc_Portale Inputs/.I_JDriveDigitalInput <-> Module 1 (Switching modes of operation)/Inputs/Digital inputs actual value
//     Plc_Portale Inputs/.I_JDriveError <-> Module 1 (Switching modes of operation)/Inputs/DriveErrorCode
//     Plc_Portale Outputs/.O_JDriveDigitalOutput <-> Module 1 (Switching modes of operation)/Outputs/CiA402 Digital outputs connector
//   PLC_Portale/PLC_Portale Instance <-> Device 3 (EtherCAT)/AsseX (MOVI-C MOVIDRIVE CiA402)
//     Plc_Portale Inputs/.I_XDriveDigitalInput <-> Module 1 (Switching modes of operation)/Inputs/Digital inputs actual value
//     Plc_Portale Inputs/.I_XDriveError <-> Module 1 (Switching modes of operation)/Inputs/DriveErrorCode
//     Plc_Portale Outputs/.O_XDriveDigitalOutput <-> Module 1 (Switching modes of operation)/Outputs/CiA402 Digital outputs connector
//   PLC_Portale/PLC_Portale Instance <-> Device 3 (EtherCAT)/AsseY (MOVI-C MOVIDRIVE CiA402)
//     Plc_Portale Inputs/.I_YDriveDigitalInput <-> Module 1 (Switching modes of operation)/Inputs/Digital inputs actual value
//     Plc_Portale Inputs/.I_YDriveError <-> Module 1 (Switching modes of operation)/Inputs/DriveErrorCode
//     Plc_Portale Outputs/.O_YDriveDigitalOutput <-> Module 1 (Switching modes of operation)/Outputs/CiA402 Digital outputs connector
//   PLC_Portale/PLC_Portale Instance <-> Device 3 (EtherCAT)/AsseZ (MOVI-C MOVIDRIVE CiA402)
//     Plc_Portale Inputs/.I_ZDriveDigitalInput <-> Module 1 (Switching modes of operation)/Inputs/Digital inputs actual value
//     Plc_Portale Inputs/.I_ZDriveError <-> Module 1 (Switching modes of operation)/Inputs/DriveErrorCode
//     Plc_Portale Outputs/.O_ZDriveDigitalOutput <-> Module 1 (Switching modes of operation)/Outputs/CiA402 Digital outputs connector
//   PLC_Portale/PLC_Portale Instance <-> Device 3 (EtherCAT)/Ciabatta IFM Pinza K515 (ifm IO-Link Master AL1332)_1
//     Plc_Portale Inputs/.I_CiabattaPinzaK515AMSADDR <-> InfoData/AdsAddr
//     Plc_Portale Inputs/.I_K515_XO3[0] <-> Module 3 (IOL_In_4Byte)/TxPDO/input byte 0
//     Plc_Portale Inputs/.I_K515_XO3[1] <-> Module 3 (IOL_In_4Byte)/TxPDO/input byte 1
//     Plc_Portale Inputs/.I_K515_XO3[2] <-> Module 3 (IOL_In_4Byte)/TxPDO/input byte 2
//     Plc_Portale Inputs/.I_K515_XO3[3] <-> Module 3 (IOL_In_4Byte)/TxPDO/input byte 3
//     Plc_Portale Inputs/.I_K515_XO4[0] <-> Module 4 (IOL_In_4Byte)/TxPDO/input byte 0
//     Plc_Portale Inputs/.I_K515_XO4[1] <-> Module 4 (IOL_In_4Byte)/TxPDO/input byte 1
//     Plc_Portale Inputs/.I_K515_XO4[2] <-> Module 4 (IOL_In_4Byte)/TxPDO/input byte 2
//     Plc_Portale Inputs/.I_K515_XO4[3] <-> Module 4 (IOL_In_4Byte)/TxPDO/input byte 3
//     Plc_Portale Inputs/.I_K517[{0..31}] <-> Module 2 (IOL_32/32_I/O-Bytes)/TxPDO/input byte {0..31}  (32 links)
//     Plc_Portale Inputs/.I_LivelloDepressioneOVEM_BH_1 <-> Module 1 (IOL_4/4_I/O-Bytes)/TxPDO/.I_LivelloDepressioneOVEM_BH_1
//     Plc_Portale Inputs/.I_LivelloDepressioneOVEM_BH_12 <-> Module 5 (IOL_4/4_I/O-Bytes)/TxPDO/.I_LivelloDepressioneOVEM_BH_12
//     Plc_Portale Inputs/.I_LivelloDepressioneOVEM_BL_1 <-> Module 1 (IOL_4/4_I/O-Bytes)/TxPDO/.I_LivelloDepressioneOVEM_BL_1
//     Plc_Portale Inputs/.I_LivelloDepressioneOVEM_BL_12 <-> Module 5 (IOL_4/4_I/O-Bytes)/TxPDO/.I_LivelloDepressioneOVEM_BL_12
//     Plc_Portale Inputs/.I_PortQualCiabattaK515_X02 <-> TxPDO IO-Link Port Qualifier/.I_PortQualCiabattaK515_X02
//     Plc_Portale Inputs/.I_PortQualCiabattaK515_X03 <-> TxPDO IO-Link Port Qualifier/.I_PortQualCiabattaK515_X03
//     Plc_Portale Inputs/.I_PortQualCiabattaK515_X04 <-> TxPDO IO-Link Port Qualifier/.I_PortQualCiabattaK515_X04
//     Plc_Portale Inputs/.I_PortQualCiabattaK515_X06 <-> TxPDO IO-Link Port Qualifier/.I_PortQualCiabattaK515_X06
//     Plc_Portale Inputs/.I_PortQualCiabattaK515_X07 <-> TxPDO IO-Link Port Qualifier/.I_PortQualCiabattaK515_X07
//     Plc_Portale Inputs/.I_PortQualCiabattaK515_X08 <-> TxPDO IO-Link Port Qualifier/.I_PortQualCiabattaK515_X08
//     Plc_Portale Inputs/.I_PortQualifierOVEM_1 <-> TxPDO IO-Link Port Qualifier/.I_PortQualifierOVEM_1
//     Plc_Portale Inputs/.I_PortQualifierOVEM_12 <-> TxPDO IO-Link Port Qualifier/.I_PortQualifierOVEM_12
//     Plc_Portale Inputs/.I_TimeStampCiabattaPinzaK515 <-> TxPDO Timestamp/.I_TimeStampCiabattaPinzaK515
//     Plc_Portale Outputs/.O_ControlWordOVEM_1 <-> Module 1 (IOL_4/4_I/O-Bytes)/RxPDO/.O_ControlWordOVEM_1
//     Plc_Portale Outputs/.O_ControlWordOVEM_12 <-> Module 5 (IOL_4/4_I/O-Bytes)/RxPDO/.O_ControlWordOVEM_12
//     Plc_Portale Outputs/.Q_K517[{0..31}] <-> Module 2 (IOL_32/32_I/O-Bytes)/RxPDO/output byte {0..31}  (32 links)
//   PLC_Portale/PLC_Portale Instance <-> Device 3 (EtherCAT)/Ciabatta IFM Pinza K516 (ifm IO-Link Master AL1332)_2
//     Plc_Portale Inputs/.I_CiabattaPinzaK516AMSADDR <-> InfoData/AdsAddr
//     Plc_Portale Inputs/.I_K516_XO3[0] <-> Module 3 (IOL_In_4Byte)/TxPDO/.I_K516_XO3[0]
//     Plc_Portale Inputs/.I_K516_XO3[1] <-> Module 3 (IOL_In_4Byte)/TxPDO/.I_K516_XO3[1]
//     Plc_Portale Inputs/.I_K516_XO3[2] <-> Module 3 (IOL_In_4Byte)/TxPDO/.I_K516_XO3[2]
//     Plc_Portale Inputs/.I_K516_XO3[3] <-> Module 3 (IOL_In_4Byte)/TxPDO/.I_K516_XO3[3]
//     Plc_Portale Inputs/.I_K516_XO4[0] <-> Module 4 (IOL_In_4Byte)/TxPDO/.I_K516_XO4[0]
//     Plc_Portale Inputs/.I_K516_XO4[1] <-> Module 4 (IOL_In_4Byte)/TxPDO/.I_K516_XO4[1]
//     Plc_Portale Inputs/.I_K516_XO4[2] <-> Module 4 (IOL_In_4Byte)/TxPDO/.I_K516_XO4[2]
//     Plc_Portale Inputs/.I_K516_XO4[3] <-> Module 4 (IOL_In_4Byte)/TxPDO/.I_K516_XO4[3]
//     Plc_Portale Inputs/.I_LivelloDepressioneOVEM_BH_2 <-> Module 1 (IOL_4/4_I/O-Bytes)/TxPDO/.I_LivelloDepressioneOVEM_BH_2
//     Plc_Portale Inputs/.I_LivelloDepressioneOVEM_BH_22 <-> Module 2 (IOL_4/4_I/O-Bytes)/TxPDO/.I_LivelloDepressioneOVEM_BH_22
//     Plc_Portale Inputs/.I_LivelloDepressioneOVEM_BL_2 <-> Module 1 (IOL_4/4_I/O-Bytes)/TxPDO/.I_LivelloDepressioneOVEM_BL_2
//     Plc_Portale Inputs/.I_LivelloDepressioneOVEM_BL_22 <-> Module 2 (IOL_4/4_I/O-Bytes)/TxPDO/.I_LivelloDepressioneOVEM_BL_22
//     Plc_Portale Inputs/.I_PortQualCiabattaK516_X03 <-> TxPDO IO-Link Port Qualifier/.I_PortQualCiabattaK516_X03
//     Plc_Portale Inputs/.I_PortQualCiabattaK516_X04 <-> TxPDO IO-Link Port Qualifier/.I_PortQualCiabattaK516_X04
//     Plc_Portale Inputs/.I_PortQualCiabattaK516_X05 <-> TxPDO IO-Link Port Qualifier/.I_PortQualCiabattaK516_X05
//     Plc_Portale Inputs/.I_PortQualCiabattaK516_X06 <-> TxPDO IO-Link Port Qualifier/.I_PortQualCiabattaK516_X06
//     Plc_Portale Inputs/.I_PortQualCiabattaK516_X07 <-> TxPDO IO-Link Port Qualifier/.I_PortQualCiabattaK516_X07
//     Plc_Portale Inputs/.I_PortQualCiabattaK516_X08 <-> TxPDO IO-Link Port Qualifier/.I_PortQualCiabattaK516_X08
//     Plc_Portale Inputs/.I_PortQualifierOVEM_2 <-> TxPDO IO-Link Port Qualifier/.I_PortQualifierOVEM_1
//     Plc_Portale Inputs/.I_PortQualifierOVEM_22 <-> TxPDO IO-Link Port Qualifier/.I_PortQualifierOVEM_2
//     Plc_Portale Inputs/.I_TimeStampCiabattaPinzaK516 <-> TxPDO Timestamp/.I_TimeStampCiabattaPinzaK516
//     Plc_Portale Outputs/.O_ControlWordOVEM_2 <-> Module 1 (IOL_4/4_I/O-Bytes)/RxPDO/.O_ControlWordOVEM_2
//     Plc_Portale Outputs/.O_ControlWordOVEM_22 <-> Module 2 (IOL_4/4_I/O-Bytes)/RxPDO/.O_ControlWordOVEM_22
//   PLC_Portale/PLC_Portale Instance <-> NC-Task 1 SAF/Axes/J
//     Plc_Portale Inputs/.J_Axis.NcToPlc <-> Outputs/ToPlc
//     Plc_Portale Outputs/.J_Axis.PlcToNc <-> Inputs/FromPlc
//   PLC_Portale/PLC_Portale Instance <-> NC-Task 1 SAF/Axes/X
//     Plc_Portale Inputs/.X_Axis.NcToPlc <-> Outputs/ToPlc
//     Plc_Portale Outputs/.X_Axis.PlcToNc <-> Inputs/FromPlc
//   PLC_Portale/PLC_Portale Instance <-> NC-Task 1 SAF/Axes/Y
//     Plc_Portale Inputs/.Y_Axis.NcToPlc <-> Outputs/ToPlc
//     Plc_Portale Outputs/.Y_Axis.PlcToNc <-> Inputs/FromPlc
//   PLC_Portale/PLC_Portale Instance <-> NC-Task 1 SAF/Axes/Z
//     Plc_Portale Inputs/.Z_Axis.NcToPlc <-> Outputs/ToPlc
//     Plc_Portale Outputs/.Z_Axis.PlcToNc <-> Inputs/FromPlc
//   (this object) <-> Device 3 (EtherCAT)/AsseX (MOVI-C MOVIDRIVE CiA402)
//     Drive/Inputs/In/nDataIn3[0] <-> Module 1 (Switching modes of operation)/Inputs/Torque actual value
//     Drive/Inputs/In/nDcOutputTime <-> InfoData/DcOutputShift
//     Drive/Inputs/In/nState1 <-> Module 1 (Switching modes of operation)/Inputs/Status word
//     Drive/Inputs/In/nState2 <-> Module 1 (Switching modes of operation)/Inputs/Status word @bit 8
//     Drive/Inputs/In/nState4 @bit 1 <-> WcState/InputToggle
//     Drive/Inputs/In/nState4 <-> WcState/WcState
//     Drive/Inputs/In/nState5 <-> Module 1 (Switching modes of operation)/Inputs/Modes of operation display
//     Drive/Outputs/Out/nCtrl1 <-> Module 1 (Switching modes of operation)/Outputs/Control word
//     Drive/Outputs/Out/nCtrl2 <-> Module 1 (Switching modes of operation)/Outputs/Control word @bit 8
//     Drive/Outputs/Out/nCtrl5 <-> Module 1 (Switching modes of operation)/Outputs/Modes of operation
//     Drive/Outputs/Out/nDataOut1 <-> Module 1 (Switching modes of operation)/Outputs/Target position
//     Drive/Outputs/Out/nDataOut2 <-> Module 1 (Switching modes of operation)/Outputs/Target velocity
//     Drive/Outputs/Out/nDataOut4[0] <-> Module 1 (Switching modes of operation)/Outputs/Target torque
//     Enc/Inputs/In/nDataIn1 <-> Module 1 (Switching modes of operation)/Inputs/Position actual value
//     Enc/Inputs/In/nDcInputTime <-> InfoData/DcInputShift
//     Enc/Inputs/In/nState4 @bit 1 <-> WcState/InputToggle
//     Enc/Inputs/In/nState4 <-> WcState/WcState
//   (this object) <-> Device 3 (EtherCAT)/AsseY (MOVI-C MOVIDRIVE CiA402)
//     Drive/Inputs/In/nDataIn3[0] <-> Module 1 (Switching modes of operation)/Inputs/Torque actual value
//     Drive/Inputs/In/nDcOutputTime <-> InfoData/DcOutputShift
//     Drive/Inputs/In/nState1 <-> Module 1 (Switching modes of operation)/Inputs/Status word
//     Drive/Inputs/In/nState2 <-> Module 1 (Switching modes of operation)/Inputs/Status word @bit 8
//     Drive/Inputs/In/nState4 @bit 1 <-> WcState/InputToggle
//     Drive/Inputs/In/nState4 <-> WcState/WcState
//     Drive/Inputs/In/nState5 <-> Module 1 (Switching modes of operation)/Inputs/Modes of operation display
//     Drive/Outputs/Out/nCtrl1 <-> Module 1 (Switching modes of operation)/Outputs/Control word
//     Drive/Outputs/Out/nCtrl2 <-> Module 1 (Switching modes of operation)/Outputs/Control word @bit 8
//     Drive/Outputs/Out/nCtrl5 <-> Module 1 (Switching modes of operation)/Outputs/Modes of operation
//     Drive/Outputs/Out/nDataOut1 <-> Module 1 (Switching modes of operation)/Outputs/Target position
//     Drive/Outputs/Out/nDataOut2 <-> Module 1 (Switching modes of operation)/Outputs/Target velocity
//     Drive/Outputs/Out/nDataOut4[0] <-> Module 1 (Switching modes of operation)/Outputs/Target torque
//     Enc/Inputs/In/nDataIn1 <-> Module 1 (Switching modes of operation)/Inputs/Position actual value
//     Enc/Inputs/In/nDcInputTime <-> InfoData/DcInputShift
//     Enc/Inputs/In/nState4 @bit 1 <-> WcState/InputToggle
//     Enc/Inputs/In/nState4 <-> WcState/WcState
//   (this object) <-> Device 3 (EtherCAT)/AsseZ (MOVI-C MOVIDRIVE CiA402)
//     Drive/Inputs/In/nDataIn3[0] <-> Module 1 (Switching modes of operation)/Inputs/Torque actual value
//     Drive/Inputs/In/nDcOutputTime <-> InfoData/DcOutputShift
//     Drive/Inputs/In/nState1 <-> Module 1 (Switching modes of operation)/Inputs/Status word
//     Drive/Inputs/In/nState2 <-> Module 1 (Switching modes of operation)/Inputs/Status word @bit 8
//     Drive/Inputs/In/nState4 @bit 1 <-> WcState/InputToggle
//     Drive/Inputs/In/nState4 <-> WcState/WcState
//     Drive/Inputs/In/nState5 <-> Module 1 (Switching modes of operation)/Inputs/Modes of operation display
//     Drive/Outputs/Out/nCtrl1 <-> Module 1 (Switching modes of operation)/Outputs/Control word
//     Drive/Outputs/Out/nCtrl2 <-> Module 1 (Switching modes of operation)/Outputs/Control word @bit 8
//     Drive/Outputs/Out/nCtrl5 <-> Module 1 (Switching modes of operation)/Outputs/Modes of operation
//     Drive/Outputs/Out/nDataOut1 <-> Module 1 (Switching modes of operation)/Outputs/Target position
//     Drive/Outputs/Out/nDataOut2 <-> Module 1 (Switching modes of operation)/Outputs/Target velocity
//     Drive/Outputs/Out/nDataOut4[0] <-> Module 1 (Switching modes of operation)/Outputs/Target torque
//     Enc/Inputs/In/nDataIn1 <-> Module 1 (Switching modes of operation)/Inputs/Position actual value
//     Enc/Inputs/In/nDcInputTime <-> InfoData/DcInputShift
//     Enc/Inputs/In/nState4 @bit 1 <-> WcState/InputToggle
//     Enc/Inputs/In/nState4 <-> WcState/WcState
//   (this object) <-> Device 3 (EtherCAT)/AsseJ (MOVI-C MOVIDRIVE CiA402)
//     Drive/Inputs/In/nDataIn3[0] <-> Module 1 (Switching modes of operation)/Inputs/Torque actual value
//     Drive/Inputs/In/nDcOutputTime <-> InfoData/DcOutputShift
//     Drive/Inputs/In/nState1 <-> Module 1 (Switching modes of operation)/Inputs/Status word
//     Drive/Inputs/In/nState2 <-> Module 1 (Switching modes of operation)/Inputs/Status word @bit 8
//     Drive/Inputs/In/nState4 @bit 1 <-> WcState/InputToggle
//     Drive/Inputs/In/nState4 <-> WcState/WcState
//     Drive/Inputs/In/nState5 <-> Module 1 (Switching modes of operation)/Inputs/Modes of operation display
//     Drive/Outputs/Out/nCtrl1 <-> Module 1 (Switching modes of operation)/Outputs/Control word
//     Drive/Outputs/Out/nCtrl2 <-> Module 1 (Switching modes of operation)/Outputs/Control word @bit 8
//     Drive/Outputs/Out/nCtrl5 <-> Module 1 (Switching modes of operation)/Outputs/Modes of operation
//     Drive/Outputs/Out/nDataOut1 <-> Module 1 (Switching modes of operation)/Outputs/Target position
//     Drive/Outputs/Out/nDataOut2 <-> Module 1 (Switching modes of operation)/Outputs/Target velocity
//     Drive/Outputs/Out/nDataOut4[0] <-> Module 1 (Switching modes of operation)/Outputs/Target torque
//     Enc/Inputs/In/nDataIn1 <-> Module 1 (Switching modes of operation)/Inputs/Position actual value
//     Enc/Inputs/In/nDcInputTime <-> InfoData/DcInputShift
//     Enc/Inputs/In/nState4 @bit 1 <-> WcState/InputToggle
//     Enc/Inputs/In/nState4 <-> WcState/WcState

CONFIGURATION PLC_Portale
    RESOURCE PLC ON TwinCAT3
        TASK Plc_Portale(INTERVAL := T#1ms, PRIORITY := 6);
        PROGRAM TFMachinePalletizerMain WITH Plc_Portale : TFMachinePalletizerMain;
    END_RESOURCE
END_CONFIGURATION

// ---- Data types/AlbertoPruevas/Enumeraciones/E_Ul_RecogidaCaballete.TcDUT

TYPE E_Ul_RecogidaCaballete :
(
	Primera_Pieza   := 0,
	LadoAMayor		:= 1,
	LadoBMayor		:= 2
);
END_TYPE

// ---- Data types/AlbertoPruevas/Estructuras/Es_FormacionCaballete/EstructuraCaballetePiking/ES_DatosPosCaballete.TcDUT
TYPE ES_DatosPosCaballetePiking :
STRUCT
	NuPiking						:UINT ;
	Lado							:UINT; 
	NumeroDePiezaPiking     		:UINT ;
	NumPosOrigenPieza				:UINT ;
	DimensionPiezaDeposito			: ES_dimensionPiezaLadoA_ladoB;
END_STRUCT
END_TYPE

// ---- Data types/AlbertoPruevas/Estructuras/Es_FormacionCaballete/EstructuraCaballetePiking/Es_PiezasCaballetePiking.TcDUT
TYPE Es_PiezasCaballetePiking :
STRUCT
	EstadoPiking			: UINT ;
	DatosPiezaPiking 		: ARRAY [1..MAXELEMENTLIST] OF ES_DatosPosCaballetePiking ;
	
	//DimensionesPiezasPiking	: ARRAY  [1..MAXELEMENTLIST] OF ES_dimensionPiezaLadoA_ladoB;
END_STRUCT
END_TYPE

// ---- Data types/AlbertoPruevas/Estructuras/Es_FormacionCaballete/Es_CoordenadasCaballeteLadoA.TcDUT
TYPE Es_CoordenadasCaballeteLadoA :
STRUCT
	CoordenadaFinale_X 							: LREAL ;
	CoordenadaFinale_Y 							: LREAL ;
	CoordenadaFinale_Z 							: LREAL ;
	CoordenadaFinale_J 							: LREAL ;
END_STRUCT
END_TYPE

// ---- Data types/AlbertoPruevas/Estructuras/Es_FormacionCaballete/Es_CoordenadasCaballeteLadoA_ladoB.TcDUT
TYPE Es_CoordenadasCaballeteLadoA_ladoB :
STRUCT
	LadoA 								: Es_CoordenadasCaballeteLadoA ;
	
	LadoB 								: Es_CoordenadasCaballeteLadoB ;
	
END_STRUCT
END_TYPE

// ---- Data types/AlbertoPruevas/Estructuras/Es_FormacionCaballete/Es_CoordenadasCaballeteLadoB.TcDUT
TYPE Es_CoordenadasCaballeteLadoB :
STRUCT
	CoordenadaFinale_X 							: LREAL ;
	CoordenadaFinale_Y 							: LREAL ;
	CoordenadaFinale_Z 							: LREAL ;
	CoordenadaFinale_J 							: LREAL ;
END_STRUCT
END_TYPE

// ---- Data types/AlbertoPruevas/Estructuras/Es_FormacionCaballete/ES_dimensionPiezaLadoA_ladoB.TcDUT
TYPE ES_dimensionPiezaLadoA_ladoB :
STRUCT
	DimPieza_LadoA 						: TFDimensionElement ;
	DimPieza_LadoB 						: TFDimensionElement ;
	Dim_Horizontal						: TFDimensionElement ;		
END_STRUCT
END_TYPE

// ---- Data types/AlbertoPruevas/Estructuras/Es_FormacionCaballete/Es_NumeroPiezasCaballete.TcDUT
TYPE Es_NumeroPiezasCaballete :
STRUCT
	Nu_Piezas_lado_A :UINT ;
	Nu_Piezas_lado_B :UINT ;
	
END_STRUCT
END_TYPE

// ---- Data types/AlbertoPruevas/Estructuras/Es_FormacionCaballete/ES_SpesoreLastra_A_B.TcDUT
TYPE ES_SpesoreLastra_A_B :
STRUCT
	Lado_A_0Grados 						: LREAL ;
	Lado_B_180Grados 					: LREAL ;
END_STRUCT
END_TYPE

// ---- Data types/AlbertoPruevas/Estructuras/Es_LadosCaballete.TcDUT
TYPE Es_LadosCaballete :
STRUCT
	Lado_trabajo 			: E_Ul_RecogidaCaballete ; // Estado del lugar Difine el estado de la rutina de descarga
	Dif_PiezasLados			: UINT ; // Contiene la diferencia de piezas entre los lados del Caballete
	TipoRecogida			: INT ; // Contine la rutina de descarga
END_STRUCT
END_TYPE

// ---- Data types/AlbertoPruevas/Estructuras/Es_PiezasCaballete.TcDUT
TYPE Es_PiezasCaballete :
STRUCT
	HMI_NumeroPezziPresentiPostazione_A_Cavaleto : UINT ;  //Numero Piezas Lado A ( 0º) caballete 
	HMI_NumeroPezziPresentiPostazione_B_Cavaleto : UINT ;  //Numero Piezas Lado B ( 180º) caballete 
	
END_STRUCT
END_TYPE

// ---- Data types/AlbertoPruevas/Estructuras/ProgramaEjecucion.TcDUT
TYPE ProgramaEjecucion :
STRUCT
	EjeX : UINT;
	EjeY : UINT;
	EjeZ : UINT;
	EjeJ : LREAL;
	CoordenadaEjeX : LREAL;
	CoordenadaEjeY : LREAL;
	CoordenadaEjeZ : LREAL;
	CoordenadaEjeJ : LREAL;
END_STRUCT
END_TYPE

// ---- Data types/DatiVari/EAP/ST_EAPAxeState.TcDUT
TYPE ST_EAPAxeState : 
	STRUCT
		(*   Actual Position mm  *)
		Position : LREAL := 0;
		(*   Actual Velocity  mm/s  *)
		Velocity : LREAL := 0;
		(*   Actual Torque   *)
		Torque : REAL := 0;
		(*   Error Code   *)
		Error : UDINT := 0;
		(*   TRUE=Power Enable   *)
		PowerActive : BOOL := false;
		(*  Home ok  *)
		Homed : BOOL := false;
	END_STRUCT
END_TYPE

// ---- Data types/DatiVari/EAP/ST_EAPCylinderState.TcDUT
TYPE ST_EAPCylinderState : 
	STRUCT
		(* Dispositivo nello stato attivo *)
		Active : BOOL;
		(* Dispositivo nello stato inattivo *)
		Inactive : BOOL;
		(* Dispositivo in errore *)
		Error : UDINT;
		(* Sensore Attivo ON *)
		SensorActive : BOOL;
		(* Senore Inattivo ON *)
		SensorInactive : BOOL;
		(* 0= Null; 1= Active ; 2= Inactive; 3= Idle; 9 = Error ; *)
		StatusToHMI : UINT;
	END_STRUCT
END_TYPE

// ---- Data types/DatiVari/EAP/ST_EAPMachineState.TcDUT
TYPE ST_EAPMachineState : 
	STRUCT
		(* Comando in esecuzione *)
		Cmd : UDINT;
		(* Stato del comando in esecuzione *)
		CmdCase : UDINT;
		(* Errore generico della Macchina *)
		Error : UDINT;
		(* Errore specifico della Macchina *)
		ErrorExtra : UDINT;
		(* Macchina con potenza attiva *)
		PowerActive : BOOL;
		(* Macchina con Home eseguito *)
		Homed : BOOL;
		(* Macchina in automatico *)
		Auto : BOOL;
		(* Macchina in automatico e con ciclo di lavoro attivo -> sta lavorando *)
		Working : BOOL;
		(* Macchina accesso manuale in area segreta attivo *)
		ManAccesActive : BOOL;
		(* Macchina in Emergenza *)
		EmergencyOK : BOOL;
	END_STRUCT
END_TYPE

// ---- Data types/DatiVari/EAP/ST_EAPModuleState.TcDUT
TYPE ST_EAPModuleState : 
	STRUCT
		(* Comando in esecuzione *)
		Cmd : UDINT;
		(* Stato del comando in esecuzione *)
		CmdCase : UDINT;
		(* Errore generico del modulo *)
		Error : UDINT;
		(* Errore specifico del modulo *)
		ErrorExtra : UDINT;
		(* Modulo in Power *)
		PowerActive : BOOL;
		(* Modulo con Home eseguito *)
		Homed : BOOL;
	END_STRUCT
END_TYPE

// ---- Data types/DatiVari/EAP/ST_EAPOvemStatus.TcDUT
TYPE ST_EAPOvemStatus : 
	STRUCT
		(*  Dispositivo Inizializzato *)
		Initialized : BOOL;
		(*  Aspirazione Attivata  *)
		Aspirazione_ON : BOOL;
		(*  Aspirazione Disattivata *)
		Aspirazione_OFF : BOOL;
		(*  Soffio Attivato *)
		Soffio_ON : BOOL;
		(*  Soffio Disattivato *)
		Soffio_OFF : BOOL;
		(*  Depressione raggiunta, data SOLO con controllo mediante comparazione interna(soglia e filtri e temporali) *)
		DepressioneSoglia_OK : BOOL;
		(* Depressione raggiunta riguardante la soglia 1 SOLO CON SOGLIE OVEM *)
		DepressioneSoglia1_OK : BOOL;
		(* Depressione raggiunta riguardante la soglia 2 SOLO CON SOGLIE OVEM *)
		DepressioneSoglia2_OK : BOOL;
		(* [mbar] Depressione Attuale *)
		ValoreDepressioneIstantanea : REAL;
		(* [mbar] Depressione Mediata su n°campioni *)
		ValoreDepressioneMediata : REAL;
		(* E' presente un errore nel modulo *)
		Error : BOOL;
		(*  Codice Errore (0=NO Errore,1=ErrMANCANZACOMUNICAZIONE,2=ErrDEVICEERROR) *)
		ErrorID : UINT;
		(*  Comando completato *)
		CommandDone : BOOL;
		(*  Errore dispositivo Resettato *)
		ErrorResetDone : BOOL;
		(*  Nessun comando attivo *)
		NoCommand_ON : BOOL;
		(*  Il dispositivo Presenta un errore *)
		DeviceError : BOOL;
		(*  Il dispositivo è disponibile/Comunica correttamente *)
		DeviceDisponibile : BOOL;
		(*  indica che è necessario effettuare la manutenzione sul dispositivo *)
		ManutenzioneNecessaria : BOOL;
		(*  indica che è il dispositivo è danneggiato *)
		GuastoDispositivo : BOOL;
		(* Indica il codice del guasto...consultare il manuale OVEM pag.24 *)
		IDGuastoDispositivo : UINT;
		(* Indica che il master non sta comunicando con il PLC *)
		ErrorMasterComunication : BOOL;
		(* Indica Chel'alimentazione dell'aria è OK	 *)
		AriaOK : BOOL;
	END_STRUCT
END_TYPE

// ---- Data types/DatiVari/EAP/ST_EAPPinzaVenstoseStateComplete.TcDUT
TYPE ST_EAPPinzaVenstoseStateComplete : 
	STRUCT
		(*   Indica che la prolunga DX della pinza è aperta   *)
		LatoDxAperto : BOOL;
		(*   Indica che la prolunga SX della pinza è aperta   *)
		LatoSxAperto : BOOL;
		(*   Indica che la prolunga DX della pinza è chiusa   *)
		LatoDxChiuso : BOOL;
		(*   Indica che la prolunga SX della pinza è chiusa   *)
		LatoSxChiuso : BOOL;
		(*   Indica che sul lato SX ho in presa la piastrella   *)
		LatoSxPiastrellaInPresa : BOOL;
		(*   Indica che sul lato DX ho in presa la piastrella   *)
		LatoDxPiastrellaInPresa : BOOL;
		(*   Indica che sul lato SX ho in presa la FALDA   *)
		LatoSxFaldaInPresa : BOOL;
		(*   Indica che sul lato DX ho in presa la FALDA   *)
		LatoDxFaldaInPresa : BOOL;
		(*   Indica che la Rotazione lungo z è sbloccata   *)
		RotazioneSbloccata : BOOL;
		(*   Indica che la rotazione lungo z è bloccata   *)
		RotazioneBloccata : BOOL;
		(*   Indica che l'elemento è stato prelevato   *)
		ElementoPrelevato : BOOL;
		(*   Indica che il piano è in presa del pezzo   *)
		PianoInPresa : BOOL;
		(*   Stato degli elementi   *)
		DeviceState : ST_EAPPinzaVentoseDeviceState;
	END_STRUCT
END_TYPE

// ---- Data types/DatiVari/EAP/ST_EAPPinzaVentoseDeviceState.TcDUT
TYPE ST_EAPPinzaVentoseDeviceState : 
	STRUCT
		(* Stato del Cilindro Apertura/chiusura pinza  *)
		CilindroApertura : ST_EAPCylinderState;
		(* Stato del Cilindro Apertura/chiusura pinza  *)
		CilindroSbloccoRotazione : ST_EAPCylinderState;
		(* Stato del Cilindro di gestione Aspirazione Falda DX *)
		AspirazioneFaldaDX : ST_EAPCylinderState;
		(* Stato del Cilindro di gestione Aspirazione Falda DX *)
		AspirazioneFaldaSX : ST_EAPCylinderState;
		(* Stato Vacuostato DX *)
		AspirazioneDX : ST_EAPOvemStatus;
		(* Stato Vacuostato SX *)
		AspirazioneSX : ST_EAPOvemStatus;
	END_STRUCT
END_TYPE

// ---- Data types/DatiVari/EAP/ST_EAPStatoPortaleVisu.TcDUT
TYPE ST_EAPStatoPortaleVisu : 
	STRUCT
		(*   X Axe State (UI Position=mm, UI Velocity=mm/sec UI Acc/Dec=mm/sec2)   *)
		AsseX : ST_EAPAxeState;
		(*   Y Axe State (UI Position=mm, UI Velocity=mm/sec UI Acc/Dec=mm/sec2)   *)
		AsseY : ST_EAPAxeState;
		(*   Z Axe State (UI Position=mm, UI Velocity=mm/sec UI Acc/Dec=mm/sec2)   *)
		AsseZ : ST_EAPAxeState;
		(*   J Axe State (UI Position=°,  UI Velocity=°/sec  UI Acc/Dec=°/sec2)   *)
		AsseJ : ST_EAPAxeState;
		(*   K Axe State (UI Position=°,  UI Velocity=°/sec  UI Acc/Dec=°/sec2)   *)
		AsseK : ST_EAPAxeState;
		(*  Stato completo della pinza  *)
		Pinza : ST_EAPPinzaVenstoseStateComplete;
		(*  Stato del modulo macchina  *)
		Macchina : ST_EAPMachineState;
		(*  Stato del modulo di gestione Asse X  *)
		ModAsse_X : ST_EAPModuleState;
		(*  Stato del modulo di gestione Asse Y  *)
		ModAsse_Y : ST_EAPModuleState;
		(*  Stato del modulo di gestione Asse z  *)
		ModAsse_Z : ST_EAPModuleState;
		(*  Stato del modulo di gestione Asse J  *)
		ModAsse_J : ST_EAPModuleState;
		(*  Stato del modulo di gestione Asse K  *)
		ModAsse_K : ST_EAPModuleState;
		(*  Stato del modulo di gestione Pinza  *)
		ModPinza : ST_EAPModuleState;
		(*  Stato del modulo di gestione Barcode  *)
		ModLettoreBc : ST_EAPModuleState;
	END_STRUCT
END_TYPE

// ---- Data types/DatiVari/e_StatoMacchinaWMS.TcDUT
{attribute 'strict'}
TYPE e_StatoMacchinaWMS :
(
	NotDefined 			:= 0,
	Allarme 			:= 3,
	ConsegnaMateriale 	:= 4,//attesa ricezione materiale da linea con ordine attivo
	Svuotamento			:= 5,
	Working 			:= 7,
	Manuale 			:= 10,
	RitiroMateriale 	:= 13,//Baie piene, attesa veicolo
	Asservimento 		:= 14	//Macchina ferma con richiesta di ingresso da veicolo
);
END_TYPE

// ---- Data types/DatiVari/e_SupportTypeAriostea.TcDUT
{attribute 'strict'}
TYPE e_SupportTypeAriostea :
(
	CAVA3100X750     := 35,		//Cavalletto	1000x3000             
	CAVA3100X740     := 37,		//Cavalletto	1500x3000             
	CSS05H150M       := 46,		//Cassa	1000x3000                  
	CSS03H120M       := 68,		//Cassa	1500x3000                  
	CSS12H120M       := 69,		//Cassa	1200x3000                  
	CAVA3370X740     := 73,		//Cavalletto	1500x3000  - 1600x3200
	CSS06H120M       := 148,	//Cassa	1500x3000  - 1600x3200     
	CAVA3100H1200    := 149 	//Cavalletto	1200x3000             
);
END_TYPE

// ---- Data types/DatiVari/ST_HskFromSupervisor.TcDUT
TYPE ST_HskFromSupervisor :
STRUCT
	(* STATO RICHIESTA VEICOLO POSTAZIONE-MACCHINA *)
	InfeedRequest			: BOOL;	// Richiesta ingresso DA LGV, TRUE= LGV è pronto per ingresso su posizione
	Encumbrance				: BOOL;	// LGV in ingombro nella postazione
	WD						: INT; 	//Whatc Dog comunicazione

   	//InfeedRequest_HW		: BOOL;	// FTC Richiesta ingresso DA LGV, TRUE = LGV è pronto per ingresso su posizione
	//OperationState 			: INT; 	// Indica il Tipo dell'operazione svolta dalla navetta: 0=Nessuna Operazione in corso
									// 1 = Prelievo in corso (valorizzato per tutta la operazione)
									// 2 = Deposito in corso (valorizzato per tutta la operazione)
	//OperationEnd 			: BOOL; // Indica la fine dell'operazione svolta dalla navetta: 1 = Operazione conclusa
									// LGV attenda la (OperationEnd_Echo)  che conferma di fine operazione da parte del PLC 
									// alla ricezione della ECHO, PC-LGV azzera : Stato Operazione =0  , Fine OPerazione =0
END_STRUCT
END_TYPE

// ---- Data types/DatiVari/ST_HskToSupervisor.TcDUT
TYPE ST_HskToSupervisor :
STRUCT
	(* STATO POSTAZIONE-MACCHINA *)
	Auto				: BOOL;	//Identifica lo stato di AUTOMATICO della macchina
	Alarm				: BOOL;	//Identifica lo stato di ERRORE della macchina
	Block				: BOOL; //Macchina-Postazione in Blocco TRUE = ogni qualvolta la macchina non può accettare il veicolo
	GateAccessActive	: BOOL; //Richiesta di ingresso manuale Operatore ATTIVATA (predisp)	
	DisableLGV			: BOOL; //Esclusione chiamata veicolo

	(* STATO CHIAMATA POSTAZIONE-MACCHINA *)
	Call_EspulsionePieno	: BOOL; // Chiamata ingresso a LGV, TRUE = La una postazione è nello stato di chiamata navetta x espulsione pieno
	Call_EspulsioneVuoto	: BOOL; // Chiamata ingresso a LGV, TRUE = La una postazione è nello stato di chiamata navetta x espulsione vuoto
	Call_RichiestoPieno		: BOOL; // Chiamata ingresso a LGV, TRUE = La una postazione è nello stato di chiamata navetta x espulsione pieno
	Call_RichiestaVuoto		: BOOL; // Chiamata ingresso a LGV, TRUE = La una postazione è nello stato di chiamata navetta x espulsione vuoto

	InfeedOK 				: BOOL; // TRUE = OK Ingresso Nella Postazione 
	
	Priority				: INT; 	//Indica la priorità di asservimento della postazione 0-100
	Saturation				: INT;	//Identifica lo stato di intasamento dei trasporti 0-100
	WD						: INT; 	//Whatc Dog comunicazione

END_STRUCT
END_TYPE

// ---- Data types/DatiVari/ST_StatisticData.TcDUT
TYPE ST_StatisticData :
STRUCT
	Auto 					: BOOL;//Automatico, tutto ok-macchina in lavoro
	Man 					: BOOL;//Manuale,non in lavoro senza errori
	Error 					: BOOL;//Macchina Ferma per qualche problema
	LGVReqEntry 			: BOOL;//Macchina in automatico con richiesta ingresso attiva
	ReadyToChange 			: BOOL;//Macchina con possibilità di eseguire il cambio
	StatoMacchina			: INT;//Stato della macchina in forma numerica: 
	TempoCicloPinza 		: ARRAY[1..4] OF INT;//Tempo ciclo di lavoro della pinza, tempo che intercorre tra prelievo-deposito-ritorno a poszione di riposo 
	PezziDepositatiActualWO : ARRAY[1..4] OF INT;//Numero di pezzi depositati ordine corrente
END_STRUCT
END_TYPE

// ---- Data types/DatiVari/ST_SupervisorData.TcDUT
TYPE ST_SupervisorData :
STRUCT
	
	HskToSupervisor 			: ST_HskToSupervisor;	//HSK da PLC a SUPERVISORE
	HskFromSupervisor 			: ST_HskFromSupervisor;	//HSK da SUPERVISORE a PLC
	DataElementToSupervisor		: ST_DataWorkArea;		//Dati elemento da PLC a SUPERVISORE
	DataElementFromSupervisor	: ST_DataWorkArea;		//Dati elemento da SUPERVISORE a PLC

END_STRUCT
END_TYPE

// ---- Data types/DatiVari/Workorder/ST_DataWorkArea.TcDUT
TYPE ST_DataWorkArea :
STRUCT
	IDWorkOrder		: LINT; (* Identificatore univoco dell'ordine di lavoro *)
	SupportType		: INT; (* Identificatore univoco supporto WMS/SUPERvISORE NAV VALORIZZA AL DEPOSITO *)
	LayerData 		: ST_LayerData; (* Identificatore/descrizione Falda WMS/SUPERvISORE NAV VALORIZZA AL DEPOSITO *)
	SlabNumber  	: INT := 0; (* Numero di lastre depositate sul supporto *)
	SlabData		: ARRAY[1..40] OF ST_SlabData; (* Sequenza delle lastre depositate *)
	Error			: INT := 0;(* Se 0=nessun errore, 1=UDC in errore -> deve andare in carwash*)
END_STRUCT
END_TYPE

// ---- Data types/DatiVari/Workorder/ST_DimensionElement.TcDUT
(* Dimensioni Elemento *)
TYPE ST_DimensionElement :
STRUCT
	XDim		: REAL	:= 0.0;	(* (mm) Dimensione X 	-> lunghezza*)
	YDim		: REAL	:= 0.0;	(* (mm) Dimensione Y  	-> larghezza *)
	ZDim		: REAL	:= 0.0;	(* (mm) Dimensione Z 	-> spessore *)
END_STRUCT
END_TYPE

// ---- Data types/DatiVari/Workorder/ST_LayerData.TcDUT
TYPE ST_LayerData :
STRUCT
	Tipologia				: INT	:= 0;  (* Indica la tipologia dell'elemento 	FALDA_CARTONE 			:= 1, (* Falde di Cartone *)
																					FALDA_POLISTIROLO 		:= 2, (* Falde di Polistirolo *)*)
	Code					: INT 	:= -1;	(* Codici del tipo falda *)
	Description				: STRING(20) := '';	(* Descrizione del tipo falda *)
	
	XDim					: REAL	:= 0.0;	(* (mm) Dimensione X -> Lunghezza *)
	YDim					: REAL	:= 0.0;	(* (mm) Dimensione Y -> Larghezza *) 
	ZDim					: REAL	:= 0.0;	(* (mm) Dimensione Z -> spessore *)
	
END_STRUCT
END_TYPE

// ---- Data types/DatiVari/Workorder/ST_SlabData.TcDUT
TYPE ST_SlabData :
STRUCT
	
	ID			: LINT := 0;		(* Unic ID - Passato da Rulliera *)
	IDWorkOrder	: LINT  := 0; 		(* Identificatore univoco dell'ordine di lavoro - Passato da Rulliera *)
	Code		: UINT  := 0;		(* Production Code - Passato da Rulliera *)
	Dimension 	: ST_DimensionElement; (* Dimensione Lastra - Passati dall'ordine *)
	DimensionReal 	: ST_DimensionElement; (* Dimensione Lastra REALI - Passati dalla RULLIERA *)
	Barcode 	: STRING(10) := ''; (* Barcode della lastra - Letto dal lettore *)
	
END_STRUCT
END_TYPE

// ---- Data types/DatiVari/Workorder/ST_SupportData.TcDUT
TYPE ST_SupportData :
STRUCT
	Tipologia				: INT	:= 0;  (* Indica la tipologia dell'elemento: 	PALLET_STANDARD 	:= 1, (* Indica la tipologia di Pallet standard *)
																					CASSA_STANDARD		:= 2,(* Indica la tipologia di cassa in legno standard *)
																					CAVALLETTO			:= 3,(* Indica la tipologia cavalletto GENERICA *)*)
																				 
	Code					: INT 	:= -1;	(* Codici Del supporto *)
	XDim					: REAL	:= 0.0;	(* (mm) Dimensione X ex Lunghezza_Cavallina*) // Lunghezza X della cavallina (Lunghezza per la cassa)
	YDim					: REAL	:= 0.0;	(* (mm) Dimensione Y ex L_Base *) // Larghezza totale della base della cavallina (Larghezza della cassa)
	ZDim					: REAL	:= 0.0;	(* (mm) Dimensione Z Base Cavallina(interno, + bassa) o Base Cassa *)
	HMAX					: REAL  := 0.0;	(* (mm) Altezza Massima dell'elemento telaio cavallina o sponde cassa, dal terreno alla massima altezza*)

	DimVertice 				: REAL  := 0.0; // Larghezza parte alta della cavallina
	DimBaseUtile 			: REAL  := 0.0; // Larghezza della base utile di appoggio delle lastre x cavallina
	
END_STRUCT
END_TYPE

// ---- Data types/DatiVari/Workorder/ST_WorkOrder.TcDUT
TYPE ST_WorkOrder :
STRUCT
	IDWorkOrder		: LINT; (* Identificatore univoco dell'ordine di lavoro *)
	State			: INT; (* Stato dell'ordine di lavoro : 1=DA ESEGUIRE,2=IN ESECUZIONE,3=TERMINATO *)
	Support			: ST_SupportData; (* Struttura descrizione supporto *)
	Layer 			: ST_LayerData; (* Struttura descrizione falda *)
	SlabNumber  	: INT; (* Numero di lastre da depositare sul supporto *)
	SlabDimension 	: ST_DimensionElement; (* Dimensione Lastra *)
	LayerSequence 	: INT; (* Sequenza di deposito delle falde -> 0=Nessuna falda,1=Deposito dopo ogni lastra,2=Deposito ogni 2 lastre,ecc*)
	ReadyToChange	: INT; (* Se = 1, la macchina è pronta a eseguire il cambio ordine *) 
END_STRUCT
END_TYPE

// ---- Data types/DatiVari/Workorder/ST_WorkOrder_Premium.TcDUT
TYPE ST_WorkOrder_Premium :
STRUCT
	IDWorkOrder		: STRING; (* Identificatore univoco dell'ordine di lavoro *)
	State			: INT; (* Stato dell'ordine di lavoro : 1=DA ESEGUIRE,2=IN ESECUZIONE,3=TERMINATO *)
	Support			: ST_SupportData; (* Struttura descrizione supporto *)
	Layer 			: ST_LayerData; (* Struttura descrizione falda *)
	SlabNumber  	: INT; (* Numero di lastre da depositare sul supporto *)
	SlabDimension 	: ST_DimensionElement; (* Dimensione Lastra *)
	LayerSequence 	: INT; (* Sequenza di deposito delle falde -> 0=Nessuna falda,1=Deposito dopo ogni lastra,2=Deposito ogni 2 lastre,ecc*)
END_STRUCT
END_TYPE

// ---- Data types/Enum/e_Disposizione_FTC_WA.TcTLEO
{attribute 'Tc2GvlVarNames'}
{attribute 'strict'}
//Disposizione Fotocellula Di Presenza in WA
TYPE e_Disposizione_FTC_WA :
(
	NOT_DEFINED			:= -1,
	FTC_PRESENZA_ANGOLO_DX	 := 1,	(* Identifica che la fotocellula di presenza della WorkArea è disposta nell'angolo a DX della WorkArea stessa *)
	FTC_PRESENZA_CENTRALE	 := 2,	(* Identifica che la fotocellula di presenza della WorkArea è disposta sulla mediana della WorkArea stessa *)	
	FTC_PRESENZA_ANGOLO_SX	 := 3	(* Identifica che la fotocellula di presenza della WorkArea è disposta nell'angolo a SX della WorkArea stessa *)
);
END_TYPE
//  NOT_DEFINED = '-1'

// ---- Data types/Enum/e_Disposizione_Postazioni.TcDUT
{attribute 'Tc2GvlVarNames'}
{attribute 'strict'}
//Disposizione delle postazioni di Prelievo/Deposito: indica in quale asse le postazioni sono disposte
TYPE e_Disposizione_Postazioni :
(
	LUNGO_X := 0, //L'asse di tutte le postazioni di Prelievo/Deposito è parallelo all'asse X della macchina
	LUNGO_Y := 1 //L'asse di tutte le postazioni di Prelievo/Deposito è ortogonale all'asse X della macchina 
);
END_TYPE
(*
*************************************************************
*                                           				*
* 		|                                   				*
*       |                                   				*
*       |                        |         |  		|		*
*       |                        |         | 		|		*
*   ----|----         ------------------------------------  *
*       |                        |         |  		|		*
*       |                        |         |  		|		*
*       |                               LUNGO X 			*
*   ----|----            					                *
*       |                                   				*
*       |                                   				*
*       |                                   				*
*   ----|----                               				*
*       |                                   				*
*       |                                   				*
*       |                                   				*	^ Y
*       |                                   				*	|
*       |                                   				*	|
*    LUNGO Y                        						*	|
*************************************************************	|
														X <-----|-
*)

// ---- Data types/Enum/e_PosizionePinza.TcDUT
{attribute 'qualified_only'}
{attribute 'strict'}
//Posizione della pinza rispetto le postazioni
TYPE e_PosizionePinza :
(
	POS_CORRIDOIO_SX 	:= 1, //La pinza si trova a SX rispetto le postazioni
	POS_CENTRALE 		:= 2, //La Pinza si trova nell'intorno del centro delle postazioni
	POS_CORRIDOIO_DX 	:= 3 //La pinza si trova a DX rispetto le postazioni
);
END_TYPE

// ---- Data types/Enum/e_RiferimentoPostazione.TcTLEO
{attribute 'Tc2GvlVarNames'}
{attribute 'strict'}
//Riferimento origine assi postazione in WA rispetto l'origine degli assi
TYPE e_RiferimentoPostazione :
(
	NOT_DEFINED			:= -1,
	ANGOLO_DX	 	:= 1,	(* Identifica che IL RISCONTRO della WorkArea è disposta nell'angolo a DX della WorkArea stessa *)
	CENTRALE	 	:= 2,	(* Identifica che IL RISCONTRO della WorkArea è disposta sulla mediana della WorkArea stessa *)	
	ANGOLO_SX	 	:= 3,	(* Identifica che IL RISCONTRO della WorkArea è disposta nell'angolo a SX della WorkArea stessa *)
	XSX_YCENTRALE 	:= 4, 	(* Identifica che IL RISCONTRO della WorkArea è disposta SX della WorkArea stessa MA LASSE Y è IN CENTRO*)
	XDX_YCENTRALE 	:= 5  	(* Identifica che IL RISCONTRO della WorkArea è disposta DX della WorkArea stessa MA LASSE Y è IN CENTRO *)
);
END_TYPE
//  NOT_DEFINED = '-1'

// ---- Data types/Enum/e_OrdinamentoPostazione.TcTLEO
{attribute 'Tc2GvlVarNames'}
{attribute 'strict'}
//Riferimento origine assi postazione in WA rispetto l'origine degli assi
TYPE e_OrdinamentoPostazione :
(
	NOT_DEFINED		:= -1,
	CRESCENTE	 	:= 1,	(* Identifica che LA numerazione CRESCE dall'origine della macchina *)
	DECRESCENTE	 	:= 2	(* Identifica che LA numerazione DECRESCE dall'origine della macchina *)	
);
END_TYPE
//  NOT_DEFINED = '-1'

// ---- Data types/Enum/e_StatoWorkOrder.TcDUT
{attribute 'qualified_only'}
{attribute 'strict'}
TYPE e_StatoWorkOrder :
(
	NON_ESEGUITO 	:= 0,
	DA_ESEGUIRE		:= 1,
	IN_ESECUZIONE 	:= 2,
	TERMINATO		:= 3
);
END_TYPE

// ---- Data types/Enum/e_Stato_Apprendimento.TcTLEO
{attribute 'Tc2GvlVarNames'}
{attribute 'strict'}
TYPE e_Stato_Apprendimento :
(
	NOT_DEFINED					:= -1,  (* Apprendimendo Indefinito *)
	APPRENDIMENTO_DISABILITATO 	:= 0, 	(* Identifica che l'apprendimento NON DEVE essere eseguito *)
	APPRENDIMENTO_DA_ESEGUIRE	:= 1, 	(* Identifica che l'apprendimento DEVE essere eseguito *)
	APPRENDIMENTO_ESEGUITO		:= 2 	(* Identifica L'AVVENUTA esecuzione dell'apprendimento*)
);
END_TYPE
//  NOT_DEFINED = '-1'

// ---- Data types/Enum/e_Stato_ElementoLista.TcTLEO
{attribute 'Tc2GvlVarNames'}
{attribute 'strict'}
//Stato dell'elemento della lista DI PRODUZIONE
TYPE e_Stato_ElementoLista :
(
	ELEMENTO_NOT_DEFINED 	:= -1, 	//STATO ELEMENTO NON DEFINITO
	ELEMENTO_DA_ELABORARE   := 0,	//STATO ELEMENTO DA ELABORARE
	ELEMENTO_ELABORATO 		:= 1 	//STATO ELEMENTO ELABORATO	
);
END_TYPE
//  ELEMENTO_NOT_DEFINED = '-1'

// ---- Data types/Enum/e_Stato_Missione.TcTLEO
{attribute 'Tc2GvlVarNames'}
{attribute 'strict'}
//Stato della Missione Della Macchina
TYPE e_Stato_Missione :
(
	NOT_DEFINED									:= -1,
	(*********************************************************************)
	MISSION_STATE_NOP							:= 0,
	(*********************************************************************)
	MISSION_STATE_INIT							:= 10,
	(*********************************************************************)
	MISSION_STATE_VAIaRIPOSO_RUN				:= 20,
	MISSION_STATE_VAIaRIPOSO_END				:= 21,
	(*********************************************************************)
	//MISSION_STATE_PRELIEVO_PALLET_RUN			:= 30,
	//MISSION_STATE_PRELIEVO_PALLET_END			:= 31,
	(*********************************************************************)
	//MISSION_STATE_DEPOSITO_PALLET_RUN			:= 40,
	//MISSION_STATE_DEPOSITO_PALLET_END			:= 41,
	(*********************************************************************)
	MISSION_STATE_PRELIEVO_FALDA_RUN			:= 50,
	MISSION_STATE_PRELIEVO_FALDA_END			:= 51,
	(*********************************************************************)
	MISSION_STATE_DEPOSITO_FALDA_RUN			:= 60,
	MISSION_STATE_DEPOSITO_FALDA_END			:= 61,
	(*********************************************************************)
//	MISSION_STATE_PRELIEVO_PACCO_RUN			:= 70,
	//MISSION_STATE_PRELIEVO_PACCO_END			:= 71,
	(*********************************************************************)
	//MISSION_STATE_DEPOSITO_PACCO_RUN			:= 80,
	//MISSION_STATE_DEPOSITO_PACCO_END			:= 81,
	(*********************************************************************)
	(*********************************************************************)
	
	MISSION_STATE_PRELIEVO_LASTRA_PP_RUN		:= 90,
	MISSION_STATE_PRELIEVO_LASTRA_PP_END		:= 91,
	(*********************************************************************)
	MISSION_STATE_DEPOSITO_LASTRA_PP_RUN		:= 100,
	MISSION_STATE_DEPOSITO_LASTRA_PP_END		:= 101,
	(*********************************************************************)
	MISSION_STATE_PRELIEVO_LASTRA_WA_RUN		:= 110,
	MISSION_STATE_PRELIEVO_LASTRA_WA_END		:= 111,
	(*********************************************************************)
	MISSION_STATE_DEPOSITO_LASTRA_WA_RUN		:= 120,
	MISSION_STATE_DEPOSITO_LASTRA_WA_END		:= 121,
	(*********************************************************************)
	MISSION_STATE_DEPOSITO_LASTRA_SU_PAREGGIATORE_RUN		:= 130,
	MISSION_STATE_DEPOSITO_LASTRA_SU_PAREGGIATORE_END		:= 131,
	(*********************************************************************)
	MISSION_STATE_PAREGGIATURA_RUN		:= 132,
	MISSION_STATE_PAREGGIATURA_END		:= 133,
	(*********************************************************************)
	MISSION_STATE_PRELIEVO_LASTRA_DA_PAREGGIATORE_RUN		:= 134,
	MISSION_STATE_PRELIEVO_LASTRA_DA_PAREGGIATORE_END		:= 135,
	(*********************************************************************)
	MISSION_STATE_PRELIEVO_LASTRA_DEPAL_RUN		:= 136,
	MISSION_STATE_PRELIEVO_LASTRA_DEPAL_END		:= 137,
	(*********************************************************************)
	MISSION_STATE_DEPOSITO_LASTRA_DEPAL_RUN	:= 138,
	MISSION_STATE_DEPOSITO_LASTRA_DEPAL_END	:= 139,
	(*********************************************************************)
	MISSION_STATE_DEPOSITO_FALDA_DEPAL_RUN	:= 140,
	MISSION_STATE_DEPOSITO_FALDA_DEPAL_END	:= 141,
	
	MISSION_STATE_ERROR							:= 999
);
END_TYPE
//  NOT_DEFINED = '-1'

// ---- Data types/Enum/e_Stato_PickPoint.TcTLEO
{attribute 'Tc2GvlVarNames'}
{attribute 'strict'}
// Stato del Punto di Prelievo 
TYPE e_Stato_PickPoint :
(
	WORKPICKPOINT_STATE_MAN			:= 0,	(* PickPoint in Stato Manuale *)
	WORKPICKPOINT_STATE_AUTO		:= 1,	(* PickPoint in Stato Automatico *)	
	WORKPICKPOINT_STATE_ERROR		:= 99 (* PickPoint in Stato di Errore *)
);
END_TYPE

// ---- Data types/Enum/e_Stato_Pareggiatura_Lastra.TcTLEO
{attribute 'Tc2GvlVarNames'}
{attribute 'strict'}
(* Pareggiatura Lastra da eseguire Prima del deposito *)
TYPE e_Stato_Pareggiatura_Lastra :
(
	PAREGGIATURA_DISABILITATA	:= 0, 
	PAREGGIATURA_DA_ESEGUIRE	:= 1, 
	PAREGGIATURA_ESEGUITA 		:= 2
);
END_TYPE

// ---- Data types/Enum/e_Stato_LetturaBarCode.TcTLEO
{attribute 'Tc2GvlVarNames'}
{attribute 'strict'}
(* Identifica lo stato della Lettura del BC:	0= Non Ancora letto/Da Leggere *)
TYPE e_Stato_LetturaBarCode :
(
	LETTURA_BC_NON_EFFETTUATA 	:= 0, // BARCODE Non Ancora letto/Da Leggere	
	LETTURA_BC_IN_CORSO			:= 1, // Lettura BARCODE In corso
	LETURA_BC_TERMINATA			:= 2, // Codice BARCODE Letto e Valido/Non da leggere, 
	LETTURA_BC_ERRATA			:= 3  // Errore durante la lettura del BARCODE 
);
END_TYPE

// ---- Data types/Enum/e_Stato_Prodotto_Su_PickPoint.TcTLEO
{attribute 'Tc2GvlVarNames'}
{attribute 'strict'}
(* Stato Prodotto Nel Pick Point *)
TYPE e_Stato_Prodotto_Su_PickPoint :
(
	WORKPICKPOINT_PRODOTTO_ASSENTE	 := 0,	(* Prodotto Presente Nel PickPoint *)
	WORKPICKPOINT_PRODOTTO_PRESENTE	 := 1	(* Prodotto Assente Nel PickPoint *)
);
END_TYPE

// ---- Data types/Enum/e_Stato_Prelievo.TcTLEO
{attribute 'Tc2GvlVarNames'}
{attribute 'strict'}
//Stato del Prelievo
TYPE e_Stato_Prelievo :
(
	PRELIEVO_NOT_DEFINED					:= -1,
	PRELIEVO_DA_EFFETTUARE		:= 0,		(* Identifica che il prelievo NON E' ancora stato EFFETTUATO *)
	PRELIEVO_EFFETTUATO			:= 1		(* Identifica che il prelievo E' STATO EFFETTUATO *)
);
END_TYPE
//  PRELIEVO_NOT_DEFINED = '-1'

// ---- Data types/Enum/e_Stato_Ingombro_EE.TcTLEO
{attribute 'Tc2GvlVarNames'}
{attribute 'strict'}
//Stato dell'ingombro dell'EndEffector
TYPE e_Stato_Ingombro_EE :
(
	EE_NOT_DEFINED				:= -1,
	EE_IN_INGOMBRO				:= 0,		(* Identifica che il Piano Di aspirazione (End-Effector) E' FUORI INGOMBRO rispetto al Punto Di prelievo *)
	EE_FUORI_INGOMBRO			:= 1		(* Identifica che il Piano Di aspirazione (End-Effector) E' IN INGOMBRO rispetto al Punto Di prelievo *)
);
END_TYPE
//  EE_NOT_DEFINED = '-1'

// ---- Data types/Enum/e_Stato_Layer.TcTLEO
{attribute 'Tc2GvlVarNames'}
{attribute 'strict'}
//Stato Deposizione Layer
TYPE e_Stato_Layer :
(
	NOT_DEFINED					:= -1,
	LAYER_DA_DEPOSITARE			:= 0, 	(* Identifica che il deposito della Falda DEVE essere eseguito *)
	LAYER_DEPOSITATO			:= 1 	(* Identifica che il deposito della Falda E' AVVENUTO o NON DEVE essere eseguito *)
);
END_TYPE
//  NOT_DEFINED = '-1'

// ---- Data types/Enum/e_Stato_Prodotto_Generico.TcTLEO
{attribute 'Tc2GvlVarNames'}
{attribute 'strict'}
(* Stato Prodotto GENERICO *)
TYPE e_Stato_Prodotto_Generico :
(
	PROD_ASSENTE	:= 0,	(* Prodotto Assente *)
	PROD_PRESENTE	:= 1	(* Prodotto Presente *)
);
END_TYPE

// ---- Data types/Enum/e_Stato_WAManager.TcTLEO
{attribute 'Tc2GvlVarNames'}
{attribute 'strict'}
//Stato del WorkAreaManager
TYPE e_Stato_WAManager :
(
	WAMANAGER_NOT_DEFINED						:= -1,
	(*********************************************************************)
	WAMANAGER_NOP								:= 100,
	(*********************************************************************)
	WAMANAGER_CICLO_RIPOSO_INIT					:= 110,
	WAMANAGER_CICLO_RIPOSO_RUN					:= 111,
	WAMANAGER_CICLO_RIPOSO_END					:= 112,
	(*********************************************************************)
	//WAMANAGER_CICLO_PALL_INIT					:= 120,
	//WAMANAGER_CICLO_PRELIEVO_PALL_RUN			:= 121,
	//WAMANAGER_CICLO_PRELIEVO_PALL_END			:= 122,
	//WAMANAGER_CICLO_DEPOSITO_PALL_RUN			:= 123,
	//WAMANAGER_CICLO_DEPOSITO_PALL_END			:= 124,
	(*********************************************************************)
	//WAMANAGER_CICLO_FALDA_VUOTI_INIT			:= 130,
	//WAMANAGER_CICLO_PRELIEVO_FALDA_VUOTI_RUN	:= 131,
	//WAMANAGER_CICLO_PRELIEVO_FALDA_VUOTI_END	:= 132,
	//WAMANAGER_CICLO_DEPOSITO_FALDA_VUOTI_RUN	:= 133,
	//WAMANAGER_CICLO_DEPOSITO_FALDA_VUOTI_END	:= 134,
	(*********************************************************************)
	WAMANAGER_CICLO_FALDA_INIT					:= 140,
	WAMANAGER_CICLO_PRELIEVO_FALDA_RUN			:= 141,
	WAMANAGER_CICLO_PRELIEVO_FALDA_END			:= 142,
	WAMANAGER_CICLO_DEPOSITO_FALDA_RUN			:= 143,
	WAMANAGER_CICLO_DEPOSITO_FALDA_END			:= 144,
	(*********************************************************************)
	//WAMANAGER_CICLO_PACCO_INIT					:= 150,
	//WAMANAGER_CICLO_PRELIEVO_PACCO_RUN			:= 151,
	//WAMANAGER_CICLO_PRELIEVO_PACCO_END			:= 152,
	//WAMANAGER_CICLO_DEPOSITO_PACCO_RUN			:= 153,
	//WAMANAGER_CICLO_DEPOSITO_PACCO_END			:= 154,
	(*********************************************************************)
	(* Ciclo Lastra NORMALE..Prelievo in Pick-Point *)
	WAMANAGER_CICLO_LASTRA_PP_INIT				:= 160, 
	WAMANAGER_CICLO_PRELIEVO_LASTRA_PP_RUN		:= 161,
	WAMANAGER_CICLO_PRELIEVO_LASTRA_PP_END		:= 162,
	WAMANAGER_CICLO_DEPOSITO_LASTRA_PP_RUN		:= 163,
	WAMANAGER_CICLO_DEPOSITO_LASTRA_PP_END		:= 164,
	(*********************************************************************)
	(* Ciclo Lastra SPECIALE..Prelievo in Work-Area *)
	WAMANAGER_CICLO_LASTRA_WA_INIT				:= 170,
	WAMANAGER_CICLO_PRELIEVO_LASTRA_WA_RUN		:= 171,
	WAMANAGER_CICLO_PRELIEVO_LASTRA_WA_END		:= 172,
	WAMANAGER_CICLO_DEPOSITO_LASTRA_WA_RUN		:= 173,
	WAMANAGER_CICLO_DEPOSITO_LASTRA_WA_END		:= 174,
	
	WAMANAGER_CICLO_DEPOSITO_LASTRA_SU_PAREGGIATORE_RUN		:= 180,
	WAMANAGER_CICLO_DEPOSITO_LASTRA_SU_PAREGGIATORE_END		:= 181,
	
	WAMANAGER_CICLO_PAREGGIATURA_RUN		:= 182,
	WAMANAGER_CICLO_PAREGGIATURA_END		:= 183,
	
	WAMANAGER_CICLO_PRELIEVO_LASTRA_DA_PAREGGIATORE_RUN		:= 184,
	WAMANAGER_CICLO_PRELIEVO_LASTRA_DA_PAREGGIATORE_END		:= 185,
	
	(* Ciclo lastra per depalettizzare da postazioni senza formature, con autoapprndimenti*)
	WAMANAGER_CICLO_LASTRA_DEPAL_INIT  			:= 190,
	WAMANAGER_CICLO_PRELIEVO_LASTRA_DEPAL_RUN	:= 191,
	WAMANAGER_CICLO_PRELIEVO_LASTRA_DEPAL_END	:= 192,
	(* Ciclo lastra deposito su rulliera *)
	WAMANAGER_CICLO_DEPOSITO_LASTRA_DEPAL_RUN	:= 193,
	WAMANAGER_CICLO_DEPOSITO_LASTRA_DEPAL_END	:= 194,
	(* Ciclo deposito FALDA su magazzino dedicato *)
	WAMANAGER_CICLO_DEPOSITO_FALDA_DEPAL_RUN 	:= 195,
	WAMANAGER_CICLO_DEPOSITO_FALDA_DEPAL_END    := 196,
	
	(*********************************************************************)	
	WAMANAGER_SALTA_DA_RIPOSO_A_PRELIEVO		:= 200
);
END_TYPE
//  WAMANAGER_NOT_DEFINED = '-1'

// ---- Data types/Enum/e_Priorita_PickPoint.TcTLEO
{attribute 'Tc2GvlVarNames'}
{attribute 'strict'}
(* Priorità Pick Point *)
TYPE e_Priorita_PickPoint :
(
	Min_PRIORITY	:= 0,	(* Pick Point con priorità Minima *)
	MAX_PRIORITY	:= 1	(* Pick Point con priorità MASSIMA *)
);
END_TYPE

// ---- Data types/Enum/e_Stato_WorkArea.TcTLEO
{attribute 'Tc2GvlVarNames'}
{attribute 'strict'}
//Stato del WorkAreaManager
TYPE e_Stato_WorkArea :
(
	WORKAREA_STATE_FREE_ENABLED					:= 0,	//WA senza pallet e Abilitata
	WORKAREA_STATE_FREE_DISABLED				:= 1,	//WA senza pallet e disabilitata
	WORKAREA_STATE_OCCUPIED_DISABLED			:= 2,	//WA con pallet e disabilitata
	WORKAREA_STATE_FREE_WORKING					:= 3,	//WA senza pallet e in lavorazione
	WORKAREA_STATE_OCCUPIED_WORKING				:= 4,	//WA con pallet e in lavorazione	
	WORKAREA_STATE_OCCUPIED_WORKED				:= 5, 	//WA con pallet e pallettizzazione terminata
	WORKAREA_STATE_OCCUPIED_WORKED_DISABLED		:= 6,	//WA con pallet e pallettizzazione terminata e area disabilitata
	WORKAREA_STATE_OCCUPIED_TAPING				:= 7,	//WA con pallet in richiesta di nastratura
	WORKAREA_STATE_OCCUPIED_TAPING_DISABLED		:= 8,	//WA con pallet in richiesta di nastratura e area disabilitata
	WORKAREA_STATE_OCCUPIED_TAPED				:= 9,	//WA con pallet e nastratura terminata
	WORKAREA_STATE_OCCUPIED_TAPED_DISABLED		:= 10,	//WA con pallet e nastratura terminata e area disabilitata
	WORKAREA_STATE_OCCUPIED_ENDED				:= 11, 	//WA con pallet e lavorazione terminata
	WORKAREA_STATE_OCCUPIED_ENDED_DISABLED		:= 12, 	//WA con pallet e lavorazione terminata e area disabilitata
	WORKAREA_STATE_OCCUPIED_LGVREQ				:= 13, 	//WA con pallet e richiesta TGV in ingresso
	WORKAREA_STATE_OCCUPIED_LGVREQ_DISABLED		:= 14, 	//WA con pallet e richiesta TGV in ingresso e area disabilitata
	WORKAREA_STATE_OCCUPIED_LGVIN				:= 15, 	//WA con pallet e TGV in ingombro
	WORKAREA_STATE_OCCUPIED_LGVIN_DISABLED		:= 16, 	//WA con pallet e TGV in ingombro e area disabilitata
	WORKAREA_STATE_OCCUPIED_LGVEND				:= 17, 	//WA con pallet e TGV fuori ingombro e Pallet estratto
	WORKAREA_STATE_OCCUPIED_LGVEND_DISABLED		:= 18, 	//WA con pallet e TGV fuori ingombro e Pallet estratto e area disabilata
	WORKAREA_STATE_OCCUPIED_LGVREQ_ABORT        := 19, 	//WA con pallet e richiesta TGV ABORTITA
	
	WORKAREA_STATE_FREE_LGVREQ					:= 20, 	//WA SENZA SUPPORTO e richiesta TGV in ingresso
	WORKAREA_STATE_FREE_LGVREQ_DISABLED			:= 21, 	//WA SENZA SUPPORTO e richiesta TGV in ingresso e area disabilitata
	WORKAREA_STATE_FREE_LGVIN					:= 22, 	//WA SENZA SUPPORTO e TGV in ingombro
	WORKAREA_STATE_FREE_LGVIN_DISABLED			:= 23, 	//WA SENZA SUPPORTO e TGV in ingombro e area disabilitata
	WORKAREA_STATE_FREE_LGVEND					:= 24, 	//WA SENZA SUPPORTO e TGV fuori ingombro e Pallet estratto
	WORKAREA_STATE_FREE_LGVEND_DISABLED			:= 25, 	//WA SENZA SUPPORTO e TGV fuori ingombro e Pallet estratto e area disabilata
	WORKAREA_STATE_FREE_LGVREQ_ABORT        	:= 26, 	//WA SENZA SUPPORTO e richiesta TGV ABORTITA
	
	WORKAREA_STATE_ERROR						:= 99	//WA in errore
);
END_TYPE

// ---- Data types/Enum/e_Stato_ListaDiProduzione.TcTLEO
{attribute 'Tc2GvlVarNames'}
{attribute 'strict'}
//Stato della lista DI PRODUZIONE
TYPE e_Stato_ListaDiProduzione :
(
	LISTA_PROD_NOT_DEFINED 		:= -1, 	//STATO LISTA PRODODUZIONE NON DEFINITO
	LISTA_PROD_ASSENTE			:= 0,	//STATO LISTA PRODODUZIONE ASSENTE:	In questo caso la macchina su questa Postazione non effettuerà alcuna lavorazione di deposito "Per composizione"
	LISTA_PROD_DA_ESEGUIRE 		:= 1, 	//STATO LISTA PRODODUZIONE DA ESEGUIRE
	LISTA_PROD_IN_ESECUZIONE 	:= 2,	//STATO LISTA PRODODUZIONE IN ESECUZIONE
	LISTA_PROD_ESEGUITA 		:= 3	//STATO LISTA PRODODUZIONE ESEGUITA
);
END_TYPE
//  LISTA_PROD_NOT_DEFINED = '-1'

// ---- Data types/Enum/e_TipologiaAreaLaser.TcDUT
{attribute 'Tc2GvlVarNames'}
{attribute 'strict'}
TYPE e_TipologiaAreaLaser :
(
	VarcoChiuso 			:= 1,
	VarcoP1_VeicoloVuoto 	:= 2,
	VarcoP1_VeicoloCarico 	:= 3,
	VarcoP2_VeicoloVuoto 	:= 4,
	VarcoP2_VeicoloCarico 	:= 5,
	VarcoP3_VeicoloVuoto 	:= 6,
	VarcoP3_VeicoloCarico 	:= 7,
	VarcoP4_VeicoloVuoto 	:= 8,
	VarcoP4_VeicoloCarico 	:= 9
	
);
END_TYPE

// ---- Data types/Enum/e_Tipologia_Rul_Prel.TcDUT
{attribute 'Tc2GvlVarNames'}
{attribute 'strict'}
//TIPOLOGIA RULLIERA DI PRELIEVO A SECONDA DI COME ARRIVA LA PIASTRELLA: 0=PUNT,1=TRAVERSO
TYPE e_Tipologia_Rul_Prel :
(
	RULLIERA_LONGITUDINALE := 0,//RULLIERA LONGITUDINALE CON ASSE X, IL PEZZO ARRIVA "DI PUNTA"
	RULLIERA_TRASVERSALE := 1 //RULLIERA TRASVERSALE CON ASSE X, IL PEZZO ARRIVA "DI TRAVERSO"
);
END_TYPE

// ---- Data types/Enum/e_Tipo_Elemento_Da_Lavorare.TcDUT
{attribute 'Tc2GvlVarNames'}
///{attribute 'strict'}
//Identifica il tipo di elemento nella tabella di 
TYPE e_Tipo_Elemento_Da_Lavorare :
(
	NOT_DEFINED				:= -1, //Elemento non definito
	LASTRA 					:= 0, //Elemento di tipo LASTRA
	FALDA					:= 1, //Elemento di tipo FALDA
	//##############################################################################################################################
	QUADROTTA 				:= 2, //Elemento di tipo "Quadrotta" ovvero, sotto prodotti che formano un piano come fosse una lastra
	//##############################################################################################################################
	TERMINATORE				:= 99 //Indica che il deposito è terminato
);

END_TYPE

// ---- Data types/Enum/e_Tipo_Magazzino_Falde.TcTLEO
{attribute 'Tc2GvlVarNames'}
{attribute 'strict'}
//Tipologia di Magazzino Falde
TYPE e_Tipo_Magazzino_Falde :
(
	NOT_DEFINED				:= -1,
	(* Magazzino Falde Per Pallettizzatore PACCHI*)
	//MAGAZZINO_FALDE_CENTRO_FISSO 		:= 1, //LA Y DI PRELIEVO RIMANE COSTANTE PER OGNI FORMATO
	//MAGAZZINO_FALDE_CENTRO_VARIABILE  	:= 2, //LA Y DI PRELIEVO SI ADATTA AL FORMATO DELLA FALDA
	
	(* Magazzino Falde per Pallettizzatore LASTRE*)
	MAGAZZINO_FALDE_IN_WA		 := 10, 	(* Identifica che il magazzino delle falde è una WorkArea *) 
	MAGAZZINO_FALDE_IN_PP		 := 20	 	(* Identifica che il magazzino delle falde è un Pick-Point, quindi elemento statico non asservito da LGV *) 

);
END_TYPE
//  NOT_DEFINED = '-1'

// ---- Data types/Enum/e_Tipo_ChiusuraAsseK.TcTLEO
{attribute 'Tc2GvlVarNames'}
{attribute 'strict'}
//Tipologia Di Presa dell' Elemento da parte dell'End Effector
TYPE e_Tipo_ChiusuraAsseK :
(
	KNOTDEFINEDMODE	:= -1,//Prelievo con ventose
	KSUCTIONMODE	:= 0,//Prelievo con ventose
	KPOSITIONMODE	:= 1,//Prelievo a quota
	KTORQUEMODE		:= 2//Prelievo con coppia
);
END_TYPE
//  KNOTDEFINEDMODE = '-1'

// ---- Data types/Enum/e_Tipo_Funzionamento.TcTLEO
{attribute 'Tc2GvlVarNames'}
{attribute 'strict'}
//Tipologia Funzionamento Macchina
TYPE e_Tipo_Funzionamento :
(
	NOT_DEFINED							:= -1, 	(* Tipologia Indefinita *)
	FUNZIONAMENTO_PALLETTIZZATORE	 	:= 0,	(* Tipologia di Funzionamento di Tipo Pallettizzatore: Prelievo Da Linea Classico *)
	FUNZIONAMENTO_PICKING				:= 1,	(* Tipologia di Funzionamento di Tipo Pallettizzatore: Prelievo e Deposito in Postazione *)
	FUNZIONAMENTO_MISTO					:= 2, 	(* Tipologia di Funzionamento di Tipo Pallettizzatore: Prelievo Da Linea Classico + Prelievo e Deposito in Postazione *)
	FUNZIONAMENTO_DEPAL					:= 3, 	(* Tipologia di Funzionamento di Tipo Depallettizzatore: Prelevo da una postazione con cavallina, cassa o pallet e appoggio sulla linea *)
	FUNZIONAMENTO_SLAVE					:= 4	(* Tipologia di Funzionamento di Tipo SLAVE: la macchina esegue le missioni che gli vengono dettate da un ente esterno (WMS)*)

);
END_TYPE
//  NOT_DEFINED = '-1'

// ---- Data types/Enum/e_Tipo_WorkArea.TcTLEO
{attribute 'Tc2GvlVarNames'}
{attribute 'strict'}
//Tipologia di WorkArea
TYPE e_Tipo_WorkArea :
(
	TYPOLOGY_NOT_DEFINED		:= -1,	(* Tipologia NON Definita *)			
	TYPOLOGY_STACK				:= 1,	(* Tipologia Catasta Vuoti *)
	TYPOLOGY_PALLET				:= 2,	(* Tipologia Postazione Di Lavoro in WorkArea *)
	TYPOLOGY_LAYER				:= 3,	(* Tipologia Postazione Magazzino Falde in WorkArea *)
	
	TYPOLOGY_OVER_TRANSPORT		:= 5,   (* Tipologia Di Postazione di prelievo/deposito su trasporti (rulliere o catenaria) *)
	TYPOLOGY_BUNDLE				:= 6,   (* Tipologia Di Postazione Di deposito = BUNDLE *)
	TYPOLOGY_ALIGNER			:= 7,   (* Tipologia Di Postazione Di PAREGGIATURA *)
	
	TYPOLOGY_WASTE				:= 8,	(* Tipologia Di Postazione SCARTI *)

	
	TYPOLOGY_EXTERNAL_DEPPREL	:= 10(* Tipologia Postazione ESTERNA al perimetro del Pallettizzatore: Utilizzata per deposito o prelievo di Pallet/Casse/Cavalline lavorate o da lavorare *)
);
END_TYPE
//  TYPOLOGY_NOT_DEFINED = '-1'

// ---- Data types/Enum/e_Tipo_Ribaltino.TcTLEO
{attribute 'Tc2GvlVarNames'}
{attribute 'strict'}
//Tipologia Ribaltino
TYPE e_Tipo_Ribaltino :
(
	RIBALTINO_NOT_DEFINED	:= -1,
	RIBALTINO_DOPO_SQUADRO  := 1, 		//Identifica il tipo di ribaltino diretto in linea, SENZA lo squadro
	RIBALTINO_DIRETTO 		:= 2 	//Identifica il tipo di ribaltino diretto in linea, SENZA lo squadro
);
END_TYPE
//  RIBALTINO_NOT_DEFINED = '-1'

// ---- Data types/Enum/e_Tipo_PickPoint.TcTLEO
{attribute 'Tc2GvlVarNames'}
{attribute 'strict'}
//Tipologia Punto DiPrelievo
TYPE e_Tipo_PickPoint :
(
	RIBALTINO_NOT_DEFINED	:= -1, (* Tipologia Indefinita *)
	RIBALTINO 				:= 1, (* Ribaltino poer pacchi classico *)
	RULLIERA				:= 2, (* Rulliera Per Lastre Classica *)
	MAGAZZINO_FALDE			:= 3, (* Magazzino Falde "Statico"*)
	

	WA_CON_CASSA			:= 4, (* Postazione in di prelievo in WorkArea in CASSA *)
	WA_CON_CAVALLINA		:= 5, (* Postazione in di prelievo in WorkArea in CAVALLINA *)
	WA_CON_PALLET			:= 6  (* Postazione di prelievo in WorkArea di tipo PALLET *)
);
END_TYPE
//  RIBALTINO_NOT_DEFINED = '-1'

// ---- Data types/Enum/e_Tipo_Falda.TcTLEO
{attribute 'Tc2GvlVarNames'}
{attribute 'strict'}
//Tipologia Falda
TYPE e_Tipo_Falda :
(
	NOT_DEFINED				:= -1,
	FALDA_CARTONE 			:= 1, (* Falde di Cartone *)
	FALDA_POLISTIROLO 		:= 2, (* Falde di Polistirolo *)
	MISTO					:= 999
);
END_TYPE
//  NOT_DEFINED = '-1'

// ---- Data types/Enum/e_Tipo_Pallet.TcTLEO
{attribute 'Tc2GvlVarNames'}
{attribute 'strict'}
//Tipologia di "Pallet/Cassa/Cavalletto" 
TYPE e_Tipo_Pallet :
(
	NOT_DEFINED			:= 0,
	PALLET_STANDARD 	:= 1, (* Indica la tipologia di Pallet standard *)
	CASSA_STANDARD		:= 2,(* Indica la tipologia di cassa in legno standard *)
	CAVALLETTO			:= 3,(* Indica la tipologia cavalletto GENERICA *)
	PALLET_ACCOPPIATI 	:= 4, (* Indica la tipologia di Pallet standard ACCOPPIATI A 2 *)
	BUNDLE				:= 5,  (* Indica la tipologia di Cavallina ad un solo lato *)
	PIANALE_GENERICO	:= 6, (* Indica un pianale generico *)
	ELEMENTO_PIANO_GENERICO := 10, (* Indica un elemento piano generico, ovvero palleto, cassa, pianale,ecc*)
	ELEMENTO_VERT_GENERICO := 11 (* Indica un elemento verticale generico, ovvero A-Frame-Bundle *)
);
END_TYPE

// ---- Data types/Enum/e_Tipo_PresaEndEffector.TcTLEO
{attribute 'Tc2GvlVarNames'}
{attribute 'strict'}
//Tipologia Di Presa dell' Elemento da parte dell'End Effector
TYPE e_Tipo_PresaEndEffector :
(
	TPICK_NOT_DEFINED							:= -1,      (* Tipo di prelievo indefinito *)
	TPICK_PACK									:= 0,		(* Identifica la presa di tipo PACCO *)
	TPICK_PALLET								:= 1,		(* Identifica la presa di tipo PALLET *)
	TPICK_LAYER									:= 2,		(* Identifica la presa di tipo FALDA (CLASSICA A VENTOSE,uitlizzata nel pal. pacchi) *)
	TPICK_LASTRA								:= 3,		(* Identifica la presa di tipo LASTRA (CLASSICA A VENTOSE) *)
	
	
	
